	HMI_ParametriAsseJ_CicloFalda.Dec_Carico 		:= HMI_ParametriAsseJ_CicloFalda.Acc_Carico;
	HMI_ParametriAsseJ_CicloFalda.Dec_Vuoto  		:= HMI_ParametriAsseJ_CicloFalda.Acc_Vuoto;
	
	HMI_ParametriAsseK_CicloFalda.Dec_Carico 		:= HMI_ParametriAsseK_CicloFalda.Acc_Carico;
	HMI_ParametriAsseK_CicloFalda.Dec_Vuoto  		:= HMI_ParametriAsseK_CicloFalda.Acc_Vuoto;
	
	(* ASSE X *)
	ParametriProgramma_X_CicloFalda.Acc_Carico		:= AxisNominalPar_X.MaximumAcceleration * (HMI_ParametriAsseX_CicloFalda.Acc_Carico/100);
	ParametriProgramma_X_CicloFalda.Acc_Vuoto		:= AxisNominalPar_X.MaximumAcceleration * (HMI_ParametriAsseX_CicloFalda.Acc_Vuoto/100);
	ParametriProgramma_X_CicloFalda.Dec_Carico 		:= AxisNominalPar_X.MaximumDeceleration * (HMI_ParametriAsseX_CicloFalda.Dec_Carico/100);
	ParametriProgramma_X_CicloFalda.Dec_Vuoto  		:= AxisNominalPar_X.MaximumDeceleration * (HMI_ParametriAsseX_CicloFalda.Dec_Vuoto/100);
	ParametriProgramma_X_CicloFalda.Jerk_Carico  	:= AxisNominalPar_X.DefaultJerk * (HMI_ParametriAsseX_CicloFalda.Jerk_Carico/100);
	ParametriProgramma_X_CicloFalda.Jerk_Vuoto  	:= AxisNominalPar_X.DefaultJerk * (HMI_ParametriAsseX_CicloFalda.Jerk_Vuoto/100);
	ParametriProgramma_X_CicloFalda.Torque  		:= AxisNominalPar_X.DefaultTorque * (HMI_ParametriAsseX_CicloFalda.Torque/100);
	ParametriProgramma_X_CicloFalda.Vel_Carico  	:= AxisNominalPar_X.ReferenceVelocity * (HMI_ParametriAsseX_CicloFalda.Vel_Carico/100) * OverrideGlobaleCicloFalda;
	ParametriProgramma_X_CicloFalda.Vel_Ridotta  	:= AxisNominalPar_X.ReferenceVelocity * (HMI_ParametriAsseX_CicloFalda.Vel_Ridotta/100);// * OverrideGlobaleCicloFalda;
	ParametriProgramma_X_CicloFalda.Vel_Vuoto  		:= AxisNominalPar_X.ReferenceVelocity * (HMI_ParametriAsseX_CicloFalda.Vel_Vuoto/100) * OverrideGlobaleCicloAvuoto;
	(* ASSE Y *)
	ParametriProgramma_Y_CicloFalda.Acc_Carico		:= AxisNominalPar_Y.MaximumAcceleration * (HMI_ParametriAsseY_CicloFalda.Acc_Carico/100);
	ParametriProgramma_Y_CicloFalda.Acc_Vuoto		:= AxisNominalPar_Y.MaximumAcceleration * (HMI_ParametriAsseY_CicloFalda.Acc_Vuoto/100);
	ParametriProgramma_Y_CicloFalda.Dec_Carico 		:= AxisNominalPar_Y.MaximumDeceleration * (HMI_ParametriAsseY_CicloFalda.Dec_Carico/100);
	ParametriProgramma_Y_CicloFalda.Dec_Vuoto  		:= AxisNominalPar_Y.MaximumDeceleration * (HMI_ParametriAsseY_CicloFalda.Dec_Vuoto/100);
	ParametriProgramma_Y_CicloFalda.Jerk_Carico  	:= AxisNominalPar_Y.DefaultJerk * (HMI_ParametriAsseY_CicloFalda.Jerk_Carico/100);
	ParametriProgramma_Y_CicloFalda.Jerk_Vuoto  	:= AxisNominalPar_Y.DefaultJerk * (HMI_ParametriAsseY_CicloFalda.Jerk_Vuoto/100);
	ParametriProgramma_Y_CicloFalda.Torque  		:= AxisNominalPar_Y.DefaultTorque * (HMI_ParametriAsseY_CicloFalda.Torque/100);
	ParametriProgramma_Y_CicloFalda.Vel_Carico  	:= AxisNominalPar_Y.ReferenceVelocity * (HMI_ParametriAsseY_CicloFalda.Vel_Carico/100) * OverrideGlobaleCicloFalda;
	ParametriProgramma_Y_CicloFalda.Vel_Ridotta  	:= AxisNominalPar_Y.ReferenceVelocity * (HMI_ParametriAsseY_CicloFalda.Vel_Ridotta/100);// * OverrideGlobaleCicloFalda;
	ParametriProgramma_Y_CicloFalda.Vel_Vuoto  		:= AxisNominalPar_Y.ReferenceVelocity * (HMI_ParametriAsseY_CicloFalda.Vel_Vuoto/100) * OverrideGlobaleCicloAvuoto;
	(* ASSE Z *)
	ParametriProgramma_Z_CicloFalda.Acc_Carico		:= AxisNominalPar_Z.MaximumAcceleration * (HMI_ParametriAsseZ_CicloFalda.Acc_Carico/100);
	ParametriProgramma_Z_CicloFalda.Acc_Vuoto		:= AxisNominalPar_Z.MaximumAcceleration * (HMI_ParametriAsseZ_CicloFalda.Acc_Vuoto/100);
	ParametriProgramma_Z_CicloFalda.Dec_Carico 		:= AxisNominalPar_Z.MaximumDeceleration * (HMI_ParametriAsseZ_CicloFalda.Dec_Carico/100);
	ParametriProgramma_Z_CicloFalda.Dec_Vuoto  		:= AxisNominalPar_Z.MaximumDeceleration * (HMI_ParametriAsseZ_CicloFalda.Dec_Vuoto/100);
	ParametriProgramma_Z_CicloFalda.Jerk_Carico  	:= AxisNominalPar_Z.DefaultJerk * (HMI_ParametriAsseZ_CicloFalda.Jerk_Carico/100);
	ParametriProgramma_Z_CicloFalda.Jerk_Vuoto  	:= AxisNominalPar_Z.DefaultJerk * (HMI_ParametriAsseZ_CicloFalda.Jerk_Vuoto/100);
	ParametriProgramma_Z_CicloFalda.Torque  		:= AxisNominalPar_Z.DefaultTorque * (HMI_ParametriAsseZ_CicloFalda.Torque/100);
	ParametriProgramma_Z_CicloFalda.Vel_Carico  	:= AxisNominalPar_Z.ReferenceVelocity * (HMI_ParametriAsseZ_CicloFalda.Vel_Carico/100) * OverrideGlobaleCicloFalda;
	ParametriProgramma_Z_CicloFalda.Vel_Ridotta  	:= AxisNominalPar_Z.ReferenceVelocity * (HMI_ParametriAsseZ_CicloFalda.Vel_Ridotta/100); //* OverrideGlobaleCicloFalda;
	ParametriProgramma_Z_CicloFalda.Vel_Vuoto  		:= AxisNominalPar_Z.ReferenceVelocity * (HMI_ParametriAsseZ_CicloFalda.Vel_Vuoto/100) * OverrideGlobaleCicloAvuoto;
	(* ASSE J *)
	ParametriProgramma_J_CicloFalda.Acc_Carico		:= AxisNominalPar_J.MaximumAcceleration * (HMI_ParametriAsseJ_CicloFalda.Acc_Carico/100);
	ParametriProgramma_J_CicloFalda.Acc_Vuoto		:= AxisNominalPar_J.MaximumAcceleration * (HMI_ParametriAsseJ_CicloFalda.Acc_Vuoto/100);
	ParametriProgramma_J_CicloFalda.Dec_Carico 		:= AxisNominalPar_J.MaximumDeceleration * (HMI_ParametriAsseJ_CicloFalda.Dec_Carico/100);
	ParametriProgramma_J_CicloFalda.Dec_Vuoto  		:= AxisNominalPar_J.MaximumDeceleration * (HMI_ParametriAsseJ_CicloFalda.Dec_Vuoto/100);
	ParametriProgramma_J_CicloFalda.Jerk_Carico  	:= AxisNominalPar_J.DefaultJerk * (HMI_ParametriAsseJ_CicloFalda.Jerk_Carico/100);
	ParametriProgramma_J_CicloFalda.Jerk_Vuoto  	:= AxisNominalPar_J.DefaultJerk * (HMI_ParametriAsseJ_CicloFalda.Jerk_Vuoto/100);
	ParametriProgramma_J_CicloFalda.Torque  		:= AxisNominalPar_J.DefaultTorque * (HMI_ParametriAsseJ_CicloFalda.Torque/100);
	ParametriProgramma_J_CicloFalda.Vel_Carico  	:= AxisNominalPar_J.ReferenceVelocity * (HMI_ParametriAsseJ_CicloFalda.Vel_Carico/100);// * OverrideGlobaleCicloFalda;
	ParametriProgramma_J_CicloFalda.Vel_Ridotta  	:= AxisNominalPar_J.ReferenceVelocity * (HMI_ParametriAsseJ_CicloFalda.Vel_Ridotta/100);// * OverrideGlobaleCicloFalda;
	ParametriProgramma_J_CicloFalda.Vel_Vuoto  		:= AxisNominalPar_J.ReferenceVelocity * (HMI_ParametriAsseJ_CicloFalda.Vel_Vuoto/100);// * OverrideGlobaleCicloAvuoto;
	(* ASSE K *)
	(*
	ParametriProgramma_K_CicloFalda.Acc_Carico		:= AxisNominalPar_K.MaximumAcceleration * (HMI_ParametriAsseK_CicloFalda.Acc_Carico/100);
	ParametriProgramma_K_CicloFalda.Acc_Vuoto		:= AxisNominalPar_K.MaximumAcceleration * (HMI_ParametriAsseK_CicloFalda.Acc_Vuoto/100);
	ParametriProgramma_K_CicloFalda.Dec_Carico 		:= AxisNominalPar_K.MaximumDeceleration * (HMI_ParametriAsseK_CicloFalda.Dec_Carico/100);
	ParametriProgramma_K_CicloFalda.Dec_Vuoto  		:= AxisNominalPar_K.MaximumDeceleration * (HMI_ParametriAsseK_CicloFalda.Dec_Vuoto/100);
	ParametriProgramma_K_CicloFalda.Jerk_Carico  	:= AxisNominalPar_K.DefaultJerk * (HMI_ParametriAsseK_CicloFalda.Jerk_Carico/100);
	ParametriProgramma_K_CicloFalda.Jerk_Vuoto  	:= AxisNominalPar_K.DefaultJerk * (HMI_ParametriAsseK_CicloFalda.Jerk_Vuoto/100);
	//ParametriProgramma_K_CicloFalda.Torque  		:= Mission^.KPickTorque;//AxisNominalPar_K.DefaultTorque * (HMI_ParametriAsseK_CicloFalda.Torque/100);
	ParametriProgramma_K_CicloFalda.Vel_Carico  	:= AxisNominalPar_K.ReferenceVelocity * (HMI_ParametriAsseK_CicloFalda.Vel_Carico/100);// * OverrideGlobaleCicloFalda;
	ParametriProgramma_K_CicloFalda.Vel_Ridotta  	:= AxisNominalPar_K.ReferenceVelocity * (HMI_ParametriAsseK_CicloFalda.Vel_Ridotta/100);// * OverrideGlobaleCicloFalda;
	ParametriProgramma_K_CicloFalda.Vel_Vuoto  		:= AxisNominalPar_K.ReferenceVelocity * (HMI_ParametriAsseK_CicloFalda.Vel_Vuoto/100);// * OverrideGlobaleCicloAvuoto;
	*)
////////////////////////////////////////////////////////////////////////////////////////////////////////////////////////////////////////////////
//////////////////////////////////////////////////// CICLO PALLET //////////////////////////////////////////////////////////////////////////////
////////////////////////////////////////////////////////////////////////////////////////////////////////////////////////////////////////////////

	HMI_ParametriAsseX_CicloPallet.Dec_Carico 		:= HMI_ParametriAsseX_CicloPallet.Acc_Carico;
	HMI_ParametriAsseX_CicloPallet.Dec_Vuoto  		:= HMI_ParametriAsseX_CicloPallet.Acc_Vuoto;

	HMI_ParametriAsseY_CicloPallet.Dec_Carico 		:= HMI_ParametriAsseY_CicloPallet.Acc_Carico;
	HMI_ParametriAsseY_CicloPallet.Dec_Vuoto  		:= HMI_ParametriAsseY_CicloPallet.Acc_Vuoto;
		
	HMI_ParametriAsseZ_CicloPallet.Dec_Carico 		:= HMI_ParametriAsseZ_CicloPallet.Acc_Carico;
	HMI_ParametriAsseZ_CicloPallet.Dec_Vuoto  		:= HMI_ParametriAsseZ_CicloPallet.Acc_Vuoto;
	
	HMI_ParametriAsseJ_CicloPallet.Dec_Carico 		:= HMI_ParametriAsseJ_CicloPallet.Acc_Carico;
	HMI_ParametriAsseJ_CicloPallet.Dec_Vuoto  		:= HMI_ParametriAsseJ_CicloPallet.Acc_Vuoto;
	
	HMI_ParametriAsseK_CicloPallet.Dec_Carico 		:= HMI_ParametriAsseK_CicloPallet.Acc_Carico;
	HMI_ParametriAsseK_CicloPallet.Dec_Vuoto  		:= HMI_ParametriAsseK_CicloPallet.Acc_Vuoto;
	
	(* ASSE X *)
	ParametriProgramma_X_CicloPallet.Acc_Carico		:= AxisNominalPar_X.MaximumAcceleration * (HMI_ParametriAsseX_CicloPallet.Acc_Carico/100);
	ParametriProgramma_X_CicloPallet.Acc_Vuoto		:= AxisNominalPar_X.MaximumAcceleration * (HMI_ParametriAsseX_CicloPallet.Acc_Vuoto/100);
	ParametriProgramma_X_CicloPallet.Dec_Carico 	:= AxisNominalPar_X.MaximumDeceleration * (HMI_ParametriAsseX_CicloPallet.Dec_Carico/100);
	ParametriProgramma_X_CicloPallet.Dec_Vuoto  	:= AxisNominalPar_X.MaximumDeceleration * (HMI_ParametriAsseX_CicloPallet.Dec_Vuoto/100);
	ParametriProgramma_X_CicloPallet.Jerk_Carico  	:= AxisNominalPar_X.DefaultJerk * (HMI_ParametriAsseX_CicloPallet.Jerk_Carico/100);
	ParametriProgramma_X_CicloPallet.Jerk_Vuoto  	:= AxisNominalPar_X.DefaultJerk * (HMI_ParametriAsseX_CicloPallet.Jerk_Vuoto/100);
	ParametriProgramma_X_CicloPallet.Torque  		:= AxisNominalPar_X.DefaultTorque * (HMI_ParametriAsseX_CicloPallet.Torque/100);
	ParametriProgramma_X_CicloPallet.Vel_Carico  	:= AxisNominalPar_X.ReferenceVelocity * (HMI_ParametriAsseX_CicloPallet.Vel_Carico/100) * OverrideGlobaleCicloPallet;
	ParametriProgramma_X_CicloPallet.Vel_Ridotta  	:= AxisNominalPar_X.ReferenceVelocity * (HMI_ParametriAsseX_CicloPallet.Vel_Ridotta/100);
	ParametriProgramma_X_CicloPallet.Vel_Vuoto  	:= AxisNominalPar_X.ReferenceVelocity * (HMI_ParametriAsseX_CicloPallet.Vel_Vuoto/100) * OverrideGlobaleCicloPallet;
	(* ASSE Y *)
	ParametriProgramma_Y_CicloPallet.Acc_Carico		:= AxisNominalPar_Y.MaximumAcceleration * (HMI_ParametriAsseY_CicloPallet.Acc_Carico/100);
	ParametriProgramma_Y_CicloPallet.Acc_Vuoto		:= AxisNominalPar_Y.MaximumAcceleration * (HMI_ParametriAsseY_CicloPallet.Acc_Vuoto/100);
	ParametriProgramma_Y_CicloPallet.Dec_Carico 	:= AxisNominalPar_Y.MaximumDeceleration * (HMI_ParametriAsseY_CicloPallet.Dec_Carico/100);
	ParametriProgramma_Y_CicloPallet.Dec_Vuoto  	:= AxisNominalPar_Y.MaximumDeceleration * (HMI_ParametriAsseY_CicloPallet.Dec_Vuoto/100);
	ParametriProgramma_Y_CicloPallet.Jerk_Carico  	:= AxisNominalPar_Y.DefaultJerk * (HMI_ParametriAsseY_CicloPallet.Jerk_Carico/100);
	ParametriProgramma_Y_CicloPallet.Jerk_Vuoto  	:= AxisNominalPar_Y.DefaultJerk * (HMI_ParametriAsseY_CicloPallet.Jerk_Vuoto/100);
	ParametriProgramma_Y_CicloPallet.Torque  		:= AxisNominalPar_Y.DefaultTorque * (HMI_ParametriAsseY_CicloPallet.Torque/100);
	ParametriProgramma_Y_CicloPallet.Vel_Carico  	:= AxisNominalPar_Y.ReferenceVelocity * (HMI_ParametriAsseY_CicloPallet.Vel_Carico/100) * OverrideGlobaleCicloPallet;
	ParametriProgramma_Y_CicloPallet.Vel_Ridotta  	:= AxisNominalPar_Y.ReferenceVelocity * (HMI_ParametriAsseY_CicloPallet.Vel_Ridotta/100);// * OverrideGlobaleCicloPallet;
	ParametriProgramma_Y_CicloPallet.Vel_Vuoto  	:= AxisNominalPar_Y.ReferenceVelocity * (HMI_ParametriAsseY_CicloPallet.Vel_Vuoto/100) * OverrideGlobaleCicloAvuoto;
	(* ASSE Z *)
	ParametriProgramma_Z_CicloPallet.Acc_Carico		:= AxisNominalPar_Z.MaximumAcceleration * (HMI_ParametriAsseZ_CicloPallet.Acc_Carico/100);
	ParametriProgramma_Z_CicloPallet.Acc_Vuoto		:= AxisNominalPar_Z.MaximumAcceleration * (HMI_ParametriAsseZ_CicloPallet.Acc_Vuoto/100);
	ParametriProgramma_Z_CicloPallet.Dec_Carico 	:= AxisNominalPar_Z.MaximumDeceleration * (HMI_ParametriAsseZ_CicloPallet.Dec_Carico/100);
	ParametriProgramma_Z_CicloPallet.Dec_Vuoto  	:= AxisNominalPar_Z.MaximumDeceleration * (HMI_ParametriAsseZ_CicloPallet.Dec_Vuoto/100);
	ParametriProgramma_Z_CicloPallet.Jerk_Carico  	:= AxisNominalPar_Z.DefaultJerk * (HMI_ParametriAsseZ_CicloPallet.Jerk_Carico/100);
	ParametriProgramma_Z_CicloPallet.Jerk_Vuoto  	:= AxisNominalPar_Z.DefaultJerk * (HMI_ParametriAsseZ_CicloPallet.Jerk_Vuoto/100);
	ParametriProgramma_Z_CicloPallet.Torque  		:= AxisNominalPar_Z.DefaultTorque * (HMI_ParametriAsseZ_CicloPallet.Torque/100);
	ParametriProgramma_Z_CicloPallet.Vel_Carico  	:= AxisNominalPar_Z.ReferenceVelocity * (HMI_ParametriAsseZ_CicloPallet.Vel_Carico/100) * OverrideGlobaleCicloPallet;
	ParametriProgramma_Z_CicloPallet.Vel_Ridotta  	:= AxisNominalPar_Z.ReferenceVelocity * (HMI_ParametriAsseZ_CicloPallet.Vel_Ridotta/100);// * OverrideGlobaleCicloPallet;
	ParametriProgramma_Z_CicloPallet.Vel_Vuoto  	:= AxisNominalPar_Z.ReferenceVelocity * (HMI_ParametriAsseZ_CicloPallet.Vel_Vuoto/100) * OverrideGlobaleCicloAvuoto;
	(* ASSE J *)
	ParametriProgramma_J_CicloPallet.Acc_Carico		:= AxisNominalPar_J.MaximumAcceleration * (HMI_ParametriAsseJ_CicloPallet.Acc_Carico/100);
	ParametriProgramma_J_CicloPallet.Acc_Vuoto		:= AxisNominalPar_J.MaximumAcceleration * (HMI_ParametriAsseJ_CicloPallet.Acc_Vuoto/100);
	ParametriProgramma_J_CicloPallet.Dec_Carico 	:= AxisNominalPar_J.MaximumDeceleration * (HMI_ParametriAsseJ_CicloPallet.Dec_Carico/100);
	ParametriProgramma_J_CicloPallet.Dec_Vuoto  	:= AxisNominalPar_J.MaximumDeceleration * (HMI_ParametriAsseJ_CicloPallet.Dec_Vuoto/100);
	ParametriProgramma_J_CicloPallet.Jerk_Carico  	:= AxisNominalPar_J.DefaultJerk * (HMI_ParametriAsseJ_CicloPallet.Jerk_Carico/100);
	ParametriProgramma_J_CicloPallet.Jerk_Vuoto  	:= AxisNominalPar_J.DefaultJerk * (HMI_ParametriAsseJ_CicloPallet.Jerk_Vuoto/100);
	ParametriProgramma_J_CicloPallet.Torque  		:= AxisNominalPar_J.DefaultTorque * (HMI_ParametriAsseJ_CicloPallet.Torque/100);
	ParametriProgramma_J_CicloPallet.Vel_Carico  	:= AxisNominalPar_J.ReferenceVelocity * (HMI_ParametriAsseJ_CicloPallet.Vel_Carico/100);// * OverrideGlobaleCicloPallet;
	ParametriProgramma_J_CicloPallet.Vel_Ridotta  	:= AxisNominalPar_J.ReferenceVelocity * (HMI_ParametriAsseJ_CicloPallet.Vel_Ridotta/100);// * OverrideGlobaleCicloPallet;
	ParametriProgramma_J_CicloPallet.Vel_Vuoto  	:= AxisNominalPar_J.ReferenceVelocity * (HMI_ParametriAsseJ_CicloPallet.Vel_Vuoto/100);// * OverrideGlobaleCicloAvuoto;
	(* ASSE K *)
	(*
	ParametriProgramma_K_CicloPallet.Acc_Carico		:= AxisNominalPar_K.MaximumAcceleration * (HMI_ParametriAsseK_CicloPallet.Acc_Carico/100);
	ParametriProgramma_K_CicloPallet.Acc_Vuoto		:= AxisNominalPar_K.MaximumAcceleration * (HMI_ParametriAsseK_CicloPallet.Acc_Vuoto/100);
	ParametriProgramma_K_CicloPallet.Dec_Carico 	:= AxisNominalPar_K.MaximumDeceleration * (HMI_ParametriAsseK_CicloPallet.Dec_Carico/100);
	ParametriProgramma_K_CicloPallet.Dec_Vuoto  	:= AxisNominalPar_K.MaximumDeceleration * (HMI_ParametriAsseK_CicloPallet.Dec_Vuoto/100);
	ParametriProgramma_K_CicloPallet.Jerk_Carico  	:= AxisNominalPar_K.DefaultJerk * (HMI_ParametriAsseK_CicloPallet.Jerk_Carico/100);
	ParametriProgramma_K_CicloPallet.Jerk_Vuoto  	:= AxisNominalPar_K.DefaultJerk * (HMI_ParametriAsseK_CicloPallet.Jerk_Vuoto/100);
	//ParametriProgramma_K_CicloPallet.Torque  		:= Mission^.KPickTorque;//AxisNominalPar_K.DefaultTorque * (HMI_ParametriAsseK_CicloPallet.Torque/100);
	ParametriProgramma_K_CicloPallet.Vel_Carico  	:= AxisNominalPar_K.ReferenceVelocity * (HMI_ParametriAsseK_CicloPallet.Vel_Carico/100);// * OverrideGlobaleCicloPallet;
	ParametriProgramma_K_CicloPallet.Vel_Ridotta  	:= AxisNominalPar_K.ReferenceVelocity * (HMI_ParametriAsseK_CicloPallet.Vel_Ridotta/100);// * OverrideGlobaleCicloPallet;
	ParametriProgramma_K_CicloPallet.Vel_Vuoto  	:= AxisNominalPar_K.ReferenceVelocity * (HMI_ParametriAsseK_CicloPallet.Vel_Vuoto/100);// * OverrideGlobaleCicloAvuoto;
	*)
////////////////////////////////////////////////////////////////////////////////////////////////////////////////////////////////////////////////
//////////////////////////////////////////////////// CICLO PACCO //////////////////////////////////////////////////////////////////////////////
////////////////////////////////////////////////////////////////////////////////////////////////////////////////////////////////////////////////


	HMI_ParametriAsseX_CicloPacco.Acc_Carico	:= MAX(1,HMI_ParametriAsseX_CicloPacco.Acc_Carico);
	HMI_ParametriAsseX_CicloPacco.Acc_Vuoto		:= MAX(1,HMI_ParametriAsseX_CicloPacco.Acc_Vuoto); 
																				 
	HMI_ParametriAsseY_CicloPacco.Acc_Carico	:= MAX(1,HMI_ParametriAsseY_CicloPacco.Acc_Carico);
	HMI_ParametriAsseY_CicloPacco.Acc_Vuoto		:= MAX(1,HMI_ParametriAsseY_CicloPacco.Acc_Vuoto); 
																				 
	HMI_ParametriAsseZ_CicloPacco.Acc_Carico	:= MAX(1,HMI_ParametriAsseZ_CicloPacco.Acc_Carico);
	HMI_ParametriAsseZ_CicloPacco.Acc_Vuoto		:= MAX(1,HMI_ParametriAsseZ_CicloPacco.Acc_Vuoto); 
																				 
	HMI_ParametriAsseJ_CicloPacco.Acc_Carico	:= MAX(1,HMI_ParametriAsseJ_CicloPacco.Acc_Carico);
	HMI_ParametriAsseJ_CicloPacco.Acc_Vuoto		:= MAX(1,HMI_ParametriAsseJ_CicloPacco.Acc_Vuoto); 
																			     
	HMI_ParametriAsseK_CicloPacco.Acc_Carico	:= MAX(1,HMI_ParametriAsseK_CicloPacco.Acc_Carico);
	HMI_ParametriAsseK_CicloPacco.Acc_Vuoto		:= MAX(1,HMI_ParametriAsseK_CicloPacco.Acc_Vuoto); 
                                                                                 
	HMI_ParametriAsseX_CicloPacco.Vel_Carico	:= MAX(1,HMI_ParametriAsseX_CicloPacco.Vel_Carico);	
	HMI_ParametriAsseX_CicloPacco.Vel_Ridotta  	:= MAX(1,HMI_ParametriAsseX_CicloPacco.Vel_Ridotta);
	

	HMI_ParametriAsseX_CicloPacco.Dec_Carico 		:= HMI_ParametriAsseX_CicloPacco.Acc_Carico;
	HMI_ParametriAsseX_CicloPacco.Dec_Vuoto  		:= HMI_ParametriAsseX_CicloPacco.Acc_Vuoto;

	HMI_ParametriAsseY_CicloPacco.Dec_Carico 		:= HMI_ParametriAsseY_CicloPacco.Acc_Carico;
	HMI_ParametriAsseY_CicloPacco.Dec_Vuoto  		:= HMI_ParametriAsseY_CicloPacco.Acc_Vuoto;
		
	HMI_ParametriAsseZ_CicloPacco.Dec_Carico 		:= HMI_ParametriAsseZ_CicloPacco.Acc_Carico;
	HMI_ParametriAsseZ_CicloPacco.Dec_Vuoto  		:= HMI_ParametriAsseZ_CicloPacco.Acc_Vuoto;
	
	HMI_ParametriAsseJ_CicloPacco.Dec_Carico 		:= HMI_ParametriAsseJ_CicloPacco.Acc_Carico;
	HMI_ParametriAsseJ_CicloPacco.Dec_Vuoto  		:= HMI_ParametriAsseJ_CicloPacco.Acc_Vuoto;
	
	HMI_ParametriAsseK_CicloPacco.Dec_Carico 		:= HMI_ParametriAsseK_CicloPacco.Acc_Carico;
	HMI_ParametriAsseK_CicloPacco.Dec_Vuoto  		:= HMI_ParametriAsseK_CicloPacco.Acc_Vuoto;

	(* ASSE X *)
	ParametriProgramma_X_CicloLastra.Acc_Carico		:= AxisNominalPar_X.MaximumAcceleration * (HMI_ParametriAsseX_CicloPacco.Acc_Carico/100);
	ParametriProgramma_X_CicloLastra.Acc_Vuoto		:= AxisNominalPar_X.MaximumAcceleration * (HMI_ParametriAsseX_CicloPacco.Acc_Vuoto/100);
	ParametriProgramma_X_CicloLastra.Dec_Carico 	:= AxisNominalPar_X.MaximumDeceleration * (HMI_ParametriAsseX_CicloPacco.Dec_Carico/100);
	ParametriProgramma_X_CicloLastra.Dec_Vuoto  	:= AxisNominalPar_X.MaximumDeceleration * (HMI_ParametriAsseX_CicloPacco.Dec_Vuoto/100);
	ParametriProgramma_X_CicloLastra.Jerk_Carico  	:= AxisNominalPar_X.DefaultJerk * (HMI_ParametriAsseX_CicloPacco.Jerk_Carico/100);
	ParametriProgramma_X_CicloLastra.Jerk_Vuoto  	:= AxisNominalPar_X.DefaultJerk * (HMI_ParametriAsseX_CicloPacco.Jerk_Vuoto/100);
	ParametriProgramma_X_CicloLastra.Torque  		:= AxisNominalPar_X.DefaultTorque * (HMI_ParametriAsseX_CicloPacco.Torque/100);
	//IF DepositoPaccoInLenta THEN
	//	ParametriProgramma_X_CicloLastra.Vel_Carico  := AxisNominalPar_X.ReferenceVelocity * (HMI_ParametriAsseX_CicloPacco.Vel_Carico/100) * OverrideGlobaleCicloPacco * (HMI_VelocitaDepositoPrimoPaccoInLenta/100);
	//ELSE
		ParametriProgramma_X_CicloLastra.Vel_Carico  := AxisNominalPar_X.ReferenceVelocity * (HMI_ParametriAsseX_CicloPacco.Vel_Carico/100) * OverrideGlobaleCicloPacco;
	//END_IF
	ParametriProgramma_X_CicloLastra.Vel_Ridotta  	:= AxisNominalPar_X.ReferenceVelocity * (HMI_ParametriAsseX_CicloPacco.Vel_Ridotta/100);// * OverrideGlobaleCicloPacco;
	ParametriProgramma_X_CicloLastra.Vel_Vuoto  		:= AxisNominalPar_X.ReferenceVelocity * (HMI_ParametriAsseX_CicloPacco.Vel_Vuoto/100) * OverrideGlobaleCicloAvuoto;
	(* ASSE Y *)
	ParametriProgramma_Y_CicloLastra.Acc_Carico		:= AxisNominalPar_Y.MaximumAcceleration * (HMI_ParametriAsseY_CicloPacco.Acc_Carico/100);
	ParametriProgramma_Y_CicloLastra.Acc_Vuoto		:= AxisNominalPar_Y.MaximumAcceleration * (HMI_ParametriAsseY_CicloPacco.Acc_Vuoto/100);
	ParametriProgramma_Y_CicloLastra.Dec_Carico 		:= AxisNominalPar_Y.MaximumDeceleration * (HMI_ParametriAsseY_CicloPacco.Dec_Carico/100);
	ParametriProgramma_Y_CicloLastra.Dec_Vuoto  		:= AxisNominalPar_Y.MaximumDeceleration * (HMI_ParametriAsseY_CicloPacco.Dec_Vuoto/100);
	ParametriProgramma_Y_CicloLastra.Jerk_Carico  	:= AxisNominalPar_Y.DefaultJerk * (HMI_ParametriAsseY_CicloPacco.Jerk_Carico/100);
	ParametriProgramma_Y_CicloLastra.Jerk_Vuoto  	:= AxisNominalPar_Y.DefaultJerk * (HMI_ParametriAsseY_CicloPacco.Jerk_Vuoto/100);
	ParametriProgramma_Y_CicloLastra.Torque  		:= AxisNominalPar_Y.DefaultTorque * (HMI_ParametriAsseY_CicloPacco.Torque/100);
	//IF DepositoPaccoInLenta THEN
	//	ParametriProgramma_Y_CicloLastra.Vel_Carico  	:= AxisNominalPar_Y.ReferenceVelocity * (HMI_ParametriAsseY_CicloPacco.Vel_Carico/100) * OverrideGlobaleCicloPacco * (HMI_VelocitaDepositoPrimoPaccoInLenta/100);
	//ELSE
		ParametriProgramma_Y_CicloLastra.Vel_Carico  	:= AxisNominalPar_Y.ReferenceVelocity * (HMI_ParametriAsseY_CicloPacco.Vel_Carico/100) * OverrideGlobaleCicloPacco;
	//END_IF
	ParametriProgramma_Y_CicloLastra.Vel_Ridotta  	:= AxisNominalPar_Y.ReferenceVelocity * (HMI_ParametriAsseY_CicloPacco.Vel_Ridotta/100);// * OverrideGlobaleCicloPacco;
	ParametriProgramma_Y_CicloLastra.Vel_Vuoto  		:= AxisNominalPar_Y.ReferenceVelocity * (HMI_ParametriAsseY_CicloPacco.Vel_Vuoto/100) * OverrideGlobaleCicloAvuoto;
	(* ASSE Z *)
	ParametriProgramma_Z_CicloLastra.Acc_Carico		:= AxisNominalPar_Z.MaximumAcceleration * (HMI_ParametriAsseZ_CicloPacco.Acc_Carico/100);
	ParametriProgramma_Z_CicloLastra.Acc_Vuoto		:= AxisNominalPar_Z.MaximumAcceleration * (HMI_ParametriAsseZ_CicloPacco.Acc_Vuoto/100);
	ParametriProgramma_Z_CicloLastra.Dec_Carico 		:= AxisNominalPar_Z.MaximumDeceleration * (HMI_ParametriAsseZ_CicloPacco.Dec_Carico/100);
	ParametriProgramma_Z_CicloLastra.Dec_Vuoto  		:= AxisNominalPar_Z.MaximumDeceleration * (HMI_ParametriAsseZ_CicloPacco.Dec_Vuoto/100);
	ParametriProgramma_Z_CicloLastra.Jerk_Carico  	:= AxisNominalPar_Z.DefaultJerk * (HMI_ParametriAsseZ_CicloPacco.Jerk_Carico/100);
	ParametriProgramma_Z_CicloLastra.Jerk_Vuoto  	:= AxisNominalPar_Z.DefaultJerk * (HMI_ParametriAsseZ_CicloPacco.Jerk_Vuoto/100);
	ParametriProgramma_Z_CicloLastra.Torque  		:= AxisNominalPar_Z.DefaultTorque * (HMI_ParametriAsseZ_CicloPacco.Torque/100);
	IF DepositoPaccoInLenta THEN
		ParametriProgramma_Z_CicloLastra.Vel_Carico  	:= AxisNominalPar_Z.ReferenceVelocity * (HMI_ParametriAsseZ_CicloPacco.Vel_Carico/100) * OverrideGlobaleCicloPacco * (HMI_VelocitaDepositoPrimoPaccoInLenta/100);
	ELSE
		ParametriProgramma_Z_CicloLastra.Vel_Carico  	:= AxisNominalPar_Z.ReferenceVelocity * (HMI_ParametriAsseZ_CicloPacco.Vel_Carico/100) * OverrideGlobaleCicloPacco;		
	END_IF
	ParametriProgramma_Z_CicloLastra.Vel_Ridotta  	:= AxisNominalPar_Z.ReferenceVelocity * (HMI_ParametriAsseZ_CicloPacco.Vel_Ridotta/100);// * OverrideGlobaleCicloPacco;
	ParametriProgramma_Z_CicloLastra.Vel_Vuoto  		:= AxisNominalPar_Z.ReferenceVelocity * (HMI_ParametriAsseZ_CicloPacco.Vel_Vuoto/100) * OverrideGlobaleCicloAvuoto;
	(* ASSE J *)
	ParametriProgramma_J_CicloLastra.Acc_Carico		:= AxisNominalPar_J.MaximumAcceleration * (HMI_ParametriAsseJ_CicloPacco.Acc_Carico/100);
	ParametriProgramma_J_CicloLastra.Acc_Vuoto		:= AxisNominalPar_J.MaximumAcceleration * (HMI_ParametriAsseJ_CicloPacco.Acc_Vuoto/100);
	ParametriProgramma_J_CicloLastra.Dec_Carico 		:= AxisNominalPar_J.MaximumDeceleration * (HMI_ParametriAsseJ_CicloPacco.Dec_Carico/100);
	ParametriProgramma_J_CicloLastra.Dec_Vuoto  		:= AxisNominalPar_J.MaximumDeceleration * (HMI_ParametriAsseJ_CicloPacco.Dec_Vuoto/100);
	ParametriProgramma_J_CicloLastra.Jerk_Carico  	:= AxisNominalPar_J.DefaultJerk * (HMI_ParametriAsseJ_CicloPacco.Jerk_Carico/100);
	ParametriProgramma_J_CicloLastra.Jerk_Vuoto  	:= AxisNominalPar_J.DefaultJerk * (HMI_ParametriAsseJ_CicloPacco.Jerk_Vuoto/100);
	ParametriProgramma_J_CicloLastra.Torque  		:= AxisNominalPar_J.DefaultTorque * (HMI_ParametriAsseJ_CicloPacco.Torque/100);
	//IF DepositoPaccoInLenta THEN
	//	ParametriProgramma_J_CicloLastra.Vel_Carico  	:= AxisNominalPar_J.ReferenceVelocity * (HMI_ParametriAsseJ_CicloPacco.Vel_Carico/100) * OverrideGlobaleCicloPacco * (HMI_VelocitaDepositoPrimoPaccoInLenta/100);
	//ELSE
		ParametriProgramma_J_CicloLastra.Vel_Carico  	:= AxisNominalPar_J.ReferenceVelocity * (HMI_ParametriAsseJ_CicloPacco.Vel_Carico/100);// * OverrideGlobaleCicloPacco;		
	//END_IF
	ParametriProgramma_J_CicloLastra.Vel_Ridotta  	:= AxisNominalPar_J.ReferenceVelocity * (HMI_ParametriAsseJ_CicloPacco.Vel_Ridotta/100);// * OverrideGlobaleCicloPacco;
	ParametriProgramma_J_CicloLastra.Vel_Vuoto  		:= AxisNominalPar_J.ReferenceVelocity * (HMI_ParametriAsseJ_CicloPacco.Vel_Vuoto/100);// * OverrideGlobaleCicloAvuoto;
	(* ASSE K *)
	(*ParametriProgramma_K_CicloLastra.Acc_Carico		:= AxisNominalPar_K.MaximumAcceleration * (HMI_ParametriAsseK_CicloPacco.Acc_Carico/100);
	ParametriProgramma_K_CicloLastra.Acc_Vuoto		:= AxisNominalPar_K.MaximumAcceleration * (HMI_ParametriAsseK_CicloPacco.Acc_Vuoto/100);
	ParametriProgramma_K_CicloLastra.Dec_Carico 		:= AxisNominalPar_K.MaximumDeceleration * (HMI_ParametriAsseK_CicloPacco.Dec_Carico/100);
	ParametriProgramma_K_CicloLastra.Dec_Vuoto  		:= AxisNominalPar_K.MaximumDeceleration * (HMI_ParametriAsseK_CicloPacco.Dec_Vuoto/100);
	ParametriProgramma_K_CicloLastra.Jerk_Carico  	:= AxisNominalPar_K.DefaultJerk * (HMI_ParametriAsseK_CicloPacco.Jerk_Carico/100);
	ParametriProgramma_K_CicloLastra.Jerk_Vuoto  	:= AxisNominalPar_K.DefaultJerk * (HMI_ParametriAsseK_CicloPacco.Jerk_Vuoto/100);
	//ParametriProgramma_K_CicloLastra.Torque  		:= Mission^.KPickTorque;//AxisNominalPar_K.DefaultTorque * (HMI_ParametriAsseK_CicloPacco.Torque/100);
	ParametriProgramma_K_CicloLastra.Vel_Carico  	:= AxisNominalPar_K.ReferenceVelocity * (HMI_ParametriAsseK_CicloPacco.Vel_Carico/100);//* OverrideGlobaleCicloPacco;
	ParametriProgramma_K_CicloLastra.Vel_Ridotta  	:= AxisNominalPar_K.ReferenceVelocity * (HMI_ParametriAsseK_CicloPacco.Vel_Ridotta/100);// * OverrideGlobaleCicloPacco;
	ParametriProgramma_K_CicloLastra.Vel_Vuoto  		:= AxisNominalPar_K.ReferenceVelocity * (HMI_ParametriAsseK_CicloPacco.Vel_Vuoto/100);//* OverrideGlobaleCicloAvuoto;
	*)

TFCalcoloVelocita := TRUE;

END_FUNCTION

// ---- POUs/TFPalletizerDataTF/TFCalcoloOverrideDinamico.TcPOU
FUNCTION TFCalcoloOverrideDinamico : REAL
VAR_INPUT
	NUltimiTrasportiOccupati : UINT;
	Overide_Dinamico : Overide_Dinamico;
END_VAR
VAR
	i : uint;
END_VAR


FOR i:= 1 TO MAXSOGLIEOVERRIDE DO
	IF NUltimiTrasportiOccupati >= Overide_Dinamico.NTrasportiOccupati[i] THEN
		TFCalcoloOverrideDinamico := Overide_Dinamico.Override[i];
		RETURN;
	END_IF
END_FOR

END_FUNCTION

// ---- POUs/TFPalletizerDataTF/TFFuoriIngombroVerticaleOK.TcPOU
FUNCTION TFFuoriIngombroVerticaleOK : BOOL
VAR_INPUT
	QuotaAsseZ : LREAL;
	Mission : POINTER TO TFMachinePalletizer_Mission;
END_VAR
VAR
END_VAR

(* Controllo Asse Z Fuori Ingombro *)
CASE Mission^.TPick OF
	TPICK_LAYER:
					IF QuotaAsseZ >= QuotaFuoriIngombro_Z_AVUOTO OR 
					QuotaAsseZ >= QuotaFuoriIngombro_Z_ConFALDA THEN
						TFFuoriIngombroVerticaleOK := TRUE;
					ELSE
						TFFuoriIngombroVerticaleOK := FALSE;
					END_IF
	TPICK_PACK :
					IF QuotaAsseZ >= QuotaFuoriIngombro_Z_AVUOTO OR 
					QuotaAsseZ >= QuotaFuoriIngombro_Z_ConPEZZO THEN
						TFFuoriIngombroVerticaleOK := TRUE;
					ELSE
						TFFuoriIngombroVerticaleOK := FALSE;
					END_IF
	TPICK_PALLET:
					IF QuotaAsseZ >= QuotaFuoriIngombro_Z_AVUOTO OR 
					QuotaAsseZ >= QuotaFuoriIngombro_Z_ConPALLET THEN
						TFFuoriIngombroVerticaleOK := TRUE;
					ELSE
						TFFuoriIngombroVerticaleOK := FALSE;
					END_IF
					
	TPICK_NOT_DEFINED:
					IF QuotaAsseZ >= QuotaFuoriIngombro_Z_AVUOTO OR 
					QuotaAsseZ >= QuotaFuoriIngombro_Z_ConPEZZO OR 
					QuotaAsseZ >= QuotaFuoriIngombro_Z_ConPALLET OR
					QuotaAsseZ >= QuotaFuoriIngombro_Z_ConFALDA THEN
						TFFuoriIngombroVerticaleOK := TRUE;
					ELSE
						TFFuoriIngombroVerticaleOK := FALSE;
					END_IF
					
	TPICK_LASTRA:
					IF QuotaAsseZ >= QuotaFuoriIngombro_Z_AVUOTO OR 
					QuotaAsseZ >= QuotaFuoriIngombro_Z_ConPEZZO THEN
						TFFuoriIngombroVerticaleOK := TRUE;
					ELSE
						TFFuoriIngombroVerticaleOK := FALSE;
					END_IF
					
	TPICK_QUADROTTA:
					IF QuotaAsseZ >= QuotaFuoriIngombro_Z_AVUOTO OR 
					QuotaAsseZ >= QuotaFuoriIngombro_Z_ConPEZZO THEN
						TFFuoriIngombroVerticaleOK := TRUE;
					ELSE
						TFFuoriIngombroVerticaleOK := FALSE;
					END_IF
					
					
					
					
					
END_CASE

END_FUNCTION

// ---- POUs/TFModules/Moduli TF/TFModulePalletizer_Aspirazione.TcPOU

FUNCTION_BLOCK TFModulePalletizer_Aspirazione
VAR_INPUT
	Cmd : CommandBuffer;
	Cfg : Config;
	IN : Module_Palletizer_Aspirazione_IN;
	
	ManCmd : Module_Palletizer_Aspirazione_ManCmd;
	
END_VAR
VAR_OUTPUT
	CmdExe : CommandExe;
	CmdExd : CommandExe;
	CmdNext : Command;
	CmdLog : CommandLog;
	ProgramLog : ProgrammaLog; 
	State : State;
	StateLog : StateLog;
	Error : Error;
	ErrorLog : ErrorLog;
	Warning : Warning;
	WarningLog : WarningLog;
	OUT : Module_Palletizer_Aspirazione_OUT;
END_VAR
VAR
	Power : UINT;
	Init : BOOL;
	Timer : REAL;
	Timeout : REAL;
	TimerAspirazione : REAL;
	ParametersArray : ParametersArray;
	MAN_Actuator : UINT;
	MAN_Cmd : UINT;
END_VAR

IF NOT Init THEN
	TFCommandBufferClear(ADR(Cmd));
	TFCommandClear(ADR(CmdNext));
	TFCommandExeClear(ADR(CmdExe));
	TFStateUpdate(ADR(State),StateNOP);
	TFErrorClear(ADR(Error));
	TFWarningClear(ADR(Warning));
	Init := TRUE;
	CmdExe.Code := 1;
END_IF

(* Generic Timer - Add here all your Timers *)
TFTimerCall(ADR(Timer),Cfg.TimeBase);
TFTimerCall(ADR(Timeout),Cfg.TimeBase);
TFTimerCall(ADR(TimerAspirazione),Cfg.TimeBase);
(* External To Buffered Command *)
TFCommandToNext(ADR(Cmd),ADR(CmdNext),ADR(CmdExe),ADR(Cfg),ADR(Error),ADR(ErrorLog),ADR(State));

(* Buffered To Exe Command *)
TFCommandToExecution(ADR(CmdNext),ADR(CmdExe),ADR(Error),ADR(ErrorLog),ADR(State),ADR(CmdLog));

(* Exe Command *)
CASE CmdExe.Code OF

	(* ******************************************************************************************************** *)
	(* Nop  *)
	(* ******************************************************************************************************** *)
	CmdNOP:	;
	
	1: TFStateUpdate(ADR(State),CmdNOP);

	(* ******************************************************************************************************** *)
	(* Stop *)
	(* ******************************************************************************************************** *)
	CmdSTOP:
		CASE CmdExe.CmdCase OF
			
			(* Case 0 *)
			0: 	TFStateUpdate(ADR(State),StateSTOP_RUN);
				TFTimerSet(ADR(Timeout),500,TRUE);
				TFCommandCase(ADR(CmdExe),1,CommandCase_INC);

			(* Case 1 - Clear All Commands*)
			1:	
				TFCommandCase(ADR(CmdExe),100,CommandCase_JMP);
			(* Case 100 *)
			100:TFStateUpdate(ADR(State),StateSTOP_END);
				TFCommandExeClear(ADR(CmdExe));

			ELSE
				TFError(ErrNOCMDCASE,ErrNULL,ADR(CmdExe),ADR(State),ADR(Error),ADR(ErrorLog));
		END_CASE;
	
	(* ******************************************************************************************************** *)
	(* Error Reset *)
	(* ******************************************************************************************************** *)
	CmdRESET:
		CASE CmdExe.CmdCase OF

			(* Case 0 *)
			0: 	TFStateUpdate(ADR(State),StateRESET_RUN);
				TFTimerSet(ADR(Timeout),2000,TRUE);
				TFCommandCase(ADR(CmdExe),1,CommandCase_INC);
			
			(* Case 1 *)
			1: TFCommandCase(ADR(CmdExe),99,CommandCase_JMP);

			
			(* Case 99 *)
			99:	TFErrorClear(ADR(Error));
				TFWarningClear(ADR(Warning));
				TFCommandCase(ADR(CmdExe),100,CommandCase_JMP);

			(* Case 100 *)
			100:TFStateUpdate(ADR(State),StateRESET_END);
				TFCommandExeClear(ADR(CmdExe));

			ELSE
				TFError(ErrNOCMDCASE,ErrNULL,ADR(CmdExe),ADR(State),ADR(Error),ADR(ErrorLog));
		END_CASE;
	
	(* ******************************************************************************************************** *)
	(* Power *)
	(* ******************************************************************************************************** *)
	CmdPOWER:
		CASE CmdExe.CmdCase OF
			
			(* Case 0 *)
			0: 	TFStateUpdate(ADR(State),StatePOWER_RUN);
				TFTimerSet(ADR(Timeout),500,TRUE);

			1: TFCommandCase(ADR(CmdExe),100,CommandCase_JMP);
			(* Case 100 *)
			100:TFStateUpdate(ADR(State),StatePOWER_END);
				TFCommandExeClear(ADR(CmdExe));

			ELSE
				TFError(ErrNOCMDCASE,ErrNULL,ADR(CmdExe),ADR(State),ADR(Error),ADR(ErrorLog));
		END_CASE
	
	(* ******************************************************************************************************** *)
	(* Home *)
	(* ******************************************************************************************************** *)
	CmdHOME:
		CASE CmdExe.CmdCase OF

			(* Case 0 *)
			0: 	TFStateUpdate(ADR(State),StateHOME_RUN);
				TFTimerSet(ADR(Timeout),30000,TRUE);
				TFCommandCase(ADR(CmdExe),1,CommandCase_INC);

			(* Case 1 - Disattivazione + Salita Ventose*)
			1: OUT.EV_Suction := FALSE;
				OUT.EV_SuctionCupsDown := FALSE;
				OUT.EV_SuctionCupsUP := TRUE;
				TFCommandCase(ADR(CmdExe),100,CommandCase_JMP);
	
			(* Case 100 *)
			100:TFStateUpdate(ADR(State),StateHOME_END);
				TFCommandExeClear(ADR(CmdExe));

			ELSE
				TFError(ErrNOCMDCASE,ErrNULL,ADR(CmdExe),ADR(State),ADR(Error),ADR(ErrorLog));
		END_CASE;

	(* ******************************************************************************************************** *)
	(* Manual *)
	(* ******************************************************************************************************** *)
	CmdMAN:
		CASE CmdExe.CmdCase OF
			(* Case 0 *)
			0: 	TFStateUpdate(ADR(State),StateMAN_RUN);
				TFTimerSet(ADR(Timeout),10,TRUE);
				IF TFCommandParRead(CmdExe.Cmd.Parameter,ADR(ParametersArray),2) THEN
					MAN_Actuator	:= STRING_TO_UINT(ParametersArray.Parameters[0]);
					MAN_Cmd		:= STRING_TO_UINT(ParametersArray.Parameters[1]);
				ELSE
					TFError(ErrCMDPARNUM,ErrNULL,ADR(CmdExe),ADR(State),ADR(Error),ADR(ErrorLog));
					RETURN;
				END_IF;

				CASE MAN_Actuator OF
					(* Case 0..99 for Actuators *)
					(* Case 100..199  for Axis *)

					(* Case Nop *)
					0:	;

					(* Case 1: *)
					1:	CASE MAN_Cmd OF
							0:	;
							
							(* Case 10: Suction OFF *)
							10:	OUT.EV_Suction := FALSE;
								
							(* Case 11: Suction ON *)
							11:	OUT.EV_Suction := TRUE;

							(* Case 10: Suction Cup Up *)
							20:	OUT.EV_SuctionCupsUp := TRUE;
								OUT.EV_SuctionCupsDown := FALSE;

							(* Case 11: Suction Cup Down *)
							21:	OUT.EV_SuctionCupsUp := FALSE;
								OUT.EV_SuctionCupsDown := TRUE;

							ELSE
								TFError(ErrNOCMDCASE,ErrNULL,ADR(CmdExe),ADR(State),ADR(Error),ADR(ErrorLog));
						END_CASE;

					100:CASE MAN_Cmd OF
							0:	;
							ELSE
								TFError(ErrNOCMDCASE,ErrNULL,ADR(CmdExe),ADR(State),ADR(Error),ADR(ErrorLog));
						END_CASE;

					ELSE
						TFError(ErrNOCMDCASE,ErrNULL,ADR(CmdExe),ADR(State),ADR(Error),ADR(ErrorLog));
				END_CASE;

				IF CmdExe.CmdCase = 0 THEN
					TFCommandCase(ADR(CmdExe),1,CommandCase_INC);
				END_IF

			(* Case 1 *)
			1: 	IF (MAN_Cmd = 0) OR TFTimerDone(ADR(Timeout)) THEN
					(* Clear All Output Here *)
					;
					TFStateUpdate(ADR(State),StateMAN_END);
					TFCommandExeClear(ADR(CmdExe));
				END_IF;
			10: ;
			(* Case 100 - End *)
			100:(* Clear All Output Here *)
				TFStateUpdate(ADR(State),StateMAN_END);
				TFCommandExeClear(ADR(CmdExe));

			ELSE
				TFError(ErrNOCMDCASE,ErrNULL,ADR(CmdExe),ADR(State),ADR(Error),ADR(ErrorLog));
		END_CASE;

	(* ******************************************************************************************************** *)
	(* LOAD - Attivazione aspirazione + discesa ventose *)
	(* ******************************************************************************************************** *)
		CmdLOAD:
		CASE CmdExe.CmdCase OF
			
			(* Case 0 - Init Command*)
			0: 	TFStateUpdate(ADR(State),StateLoad_RUN);
				TFTimerSet(ADR(Timeout),60000,TRUE);
				TFCommandCase(ADR(CmdExe),1,CommandCase_INC);
				
			(* Case 1 - Attivazione Ventosa *)					
			1:
				OUT.EV_Suction := TRUE;
				TFCommandCase(ADR(CmdExe),1,CommandCase_INC);
			(* Case 2 - Discesa Ventose *)		
			2: 
				OUT.EV_SuctionCupsDOWN 	:= TRUE;
				OUT.EV_SuctionCupsUP 	:= FALSE;
				TFTimerSet(ADR(TimerAspirazione),2000,TRUE);
				TFCommandCase(ADR(CmdExe),1,CommandCase_INC);
			3:
				IF TFTimerDone(ADR(TimerAspirazione)) THEN
					TFCommandCase(ADR(CmdExe),100,CommandCase_JMP);
				END_IF
				
			(* Case 100 *)
			100:TFStateUpdate(ADR(State),StateLOAD_END);
				TFCommandExeClear(ADR(CmdExe));

			ELSE
				TFError(ErrNOCMDCASE,ErrNULL,ADR(CmdExe),ADR(State),ADR(Error),ADR(ErrorLog));
		END_CASE
		
	(* ******************************************************************************************************** *)
	(* UNLOAD - Attivazione aspirazione + discesa ventose *)
	(* ******************************************************************************************************** *)
		CmdUNLOAD:
		CASE CmdExe.CmdCase OF
			
			(* Case 0 - Init Command*)
			0: 	TFStateUpdate(ADR(State),StateUNLOAD_RUN);
				TFTimerSet(ADR(Timeout),60000,TRUE);
				TFCommandCase(ADR(CmdExe),1,CommandCase_INC);
				
			(* Case 1 - Disattivazione Aspirazione*)					
			1:	
				OUT.EV_Suction := False;
				TFCommandCase(ADR(CmdExe),1,CommandCase_INC);
			
			(* Case 2 - Salita Ventose *)		
			2: 
				OUT.EV_SuctionCupsDOWN 	:= FALSE;
				OUT.EV_SuctionCupsUP 	:= TRUE;
				TFCommandCase(ADR(CmdExe),100,CommandCase_JMP);	
				
			(* Case 100 *)
			100:TFStateUpdate(ADR(State),StateUNLOAD_END);
				TFCommandExeClear(ADR(CmdExe));

			ELSE
				TFError(ErrNOCMDCASE,ErrNULL,ADR(CmdExe),ADR(State),ADR(Error),ADR(ErrorLog));
		END_CASE
	ELSE
		TFError(ErrNOCMD,ErrNULL,ADR(CmdExe),ADR(State),ADR(Error),ADR(ErrorLog));

END_CASE;


(* ******************************************************************************************************** *)
(* State Input/Output *)
(* ******************************************************************************************************** *)
(* Fill Input/Output bit with sensor, electrovalve, etc. status *)


(* ******************************************************************************************************** *)
(* Input *)
(* ******************************************************************************************************** *)

(* ******************************************************************************************************** *)
(* Alarm *)
(* ******************************************************************************************************** *)

(* ******************************************************************************************************** *)
(* Error Check - Clear All Output!!! *)
(* ******************************************************************************************************** *)
IF Error.Code > ErrNULL THEN
	IF CmdExe.Code <> CmdNOP THEN
		IF CmdExe.Code <> CmdSTOP AND
			CmdExe.Code <> CmdPOWER AND
			CmdExe.Code <> CmdRESET AND
			CmdExe.Code <> CmdMAN AND
			CmdExe.Code <> CmdLOAD AND
			CmdExe.Code <> CmdUNLOAD THEN
			TFCommandClear(ADR(CmdNext));
			TFCommandExeClear(ADR(CmdExe));

			(* Clear All Output Here *)

		END_IF;
	END_IF;
END_IF;


(* ******************************************************************************************************** *)
(* Common Outputs *)
(* ******************************************************************************************************** *)

END_FUNCTION_BLOCK

// ---- Data types/AlbertoPruevas/BloqueFunciones/Fb_SensoresTasteggio.TcPOU
FUNCTION_BLOCK Fb_SensoresTasteggio
VAR_INPUT
	Sensor_Tasteo_1 				: BOOL ;
	Sensor_Tasteo_2 				: BOOL ;
	Sensor_Tasteo_3 				: BOOL ;
	Sensor_Tasteo_4 				: BOOL ;
	Nu_sensores_Dar_Out				: BYTE ;
END_VAR
VAR_OUTPUT
	Sensores_Tasteggio_Ok 			: BOOL ;
	Nu_Sesores_Activos				: BYTE ;
END_VAR
VAR
END_VAR

Nu_Sesores_Activos := BOOL_TO_BYTE(Sensor_Tasteo_1) + BOOL_TO_BYTE(Sensor_Tasteo_2) + BOOL_TO_BYTE(Sensor_Tasteo_3) + BOOL_TO_BYTE(Sensor_Tasteo_4) ; 

IF Nu_Sesores_Activos >= Nu_sensores_Dar_Out THEN
	Sensores_Tasteggio_Ok := TRUE ;
	ELSE
	Sensores_Tasteggio_Ok := FALSE ;	
	
END_IF

END_FUNCTION_BLOCK

// ---- Data types/AlbertoPruevas/Funciones/FuncionesFormaciones/Fun_CalculoCoordenadasFinalesFormacion.TcPOU
FUNCTION Fun_CalculoCoordenadasFinalesFormacion : bool
VAR_INPUT
	TipoCalForCavallete 		: UINT ;
	numeroLastre_int 		: UINT ;
	Supporto 				: POINTER TO TFMachinePalletizer_Pallet;
	XFinale 				: POINTER TO  ARRAY [1..MAXFORMINGSLAB] OF LREAL;
	YFinale 				: POINTER TO  ARRAY [1..MAXFORMINGSLAB] OF LREAL;
	YInternoLastra 			: POINTER TO  ARRAY [1..MAXFORMINGSLAB] OF LREAL;
	ZFinale 				: POINTER TO  ARRAY [1..MAXFORMINGSLAB] OF LREAL;
	ZInternoLastra			: POINTER TO  ARRAY [1..MAXFORMINGSLAB] OF LREAL;
	JFinale 				: POINTER TO  ARRAY [1..MAXFORMINGSLAB] OF LREAL;
END_VAR
VAR
	Contador: UINT;
END_VAR

FOR Contador := 1 TO numeroLastre_int * 2 DO 
	CASE TipoCalForCavallete OF 
		1: 

			XFinale^[Contador] := Supporto^.XDim/2 + Supporto^.OFSDE_X180;
			;
		2: 
			;
		3:
			;
		4: 
			;
	END_CASE
	
END_FOR

END_FUNCTION

// ---- POUs/Check/CheckBounds.TcPOU
// Implicitly generated code : DO NOT EDIT
FUNCTION CheckBounds : DINT
VAR_INPUT
	index, lower, upper: DINT;
END_VAR

// Implicitly generated code : Only an Implementation suggestion
{noflow}
IF  index < lower THEN
	CheckBounds := lower;
ELSIF  index > upper THEN
	CheckBounds := upper;
ELSE  
	CheckBounds := index;
END_IF
{flow}

END_FUNCTION

// ---- POUs/Check/CheckDivDInt.TcPOU
// Implicitly generated code : DO NOT EDIT
FUNCTION CheckDivDInt : DINT
VAR_INPUT
	divisor:DINT;
END_VAR

// Implicitly generated code : Only an Implementation suggestion
{noflow}
IF divisor = 0 THEN
	CheckDivDInt:=1;
ELSE
	CheckDivDInt:=divisor;
END_IF;
{flow}

END_FUNCTION

// ---- POUs/Check/CheckDivLInt.TcPOU
// Implicitly generated code : DO NOT EDIT
FUNCTION CheckDivLInt : LINT
VAR_INPUT
	divisor:LINT;
END_VAR

// Implicitly generated code : Only an Implementation suggestion
{noflow}
IF divisor = 0 THEN
	CheckDivLInt:=1;
ELSE
	CheckDivLInt:=divisor;
END_IF;
{flow}

END_FUNCTION

// ---- POUs/Check/CheckDivLReal.TcPOU
// Implicitly generated code : DO NOT EDIT
FUNCTION CheckDivLReal : LREAL
VAR_INPUT
	divisor:LREAL;
END_VAR

// Implicitly generated code : Only an Implementation suggestion
{noflow}
IF divisor = 0 THEN
	CheckDivLReal:=1;
ELSE
	CheckDivLReal:=divisor;
END_IF;
{flow}

END_FUNCTION

// ---- POUs/Check/CheckDivReal.TcPOU
// Implicitly generated code : DO NOT EDIT
FUNCTION CheckDivReal : REAL
VAR_INPUT
	divisor:REAL;
END_VAR

// Implicitly generated code : Only an Implementation suggestion
{noflow}
IF divisor = 0 THEN
	CheckDivReal:=1;
ELSE
	CheckDivReal:=divisor;
END_IF;
{flow}

END_FUNCTION

// ---- POUs/Check/CheckLRangeSigned.TcPOU
// Implicitly generated code : DO NOT EDIT
FUNCTION CheckLRangeSigned : LINT
VAR_INPUT
	value, lower, upper: LINT;
END_VAR

// Implicitly generated code : Only an Implementation suggestion
{noflow}
IF (value < lower) THEN
	CheckLRangeSigned := lower;
ELSIF(value > upper) THEN
	CheckLRangeSigned := upper;
ELSE
	CheckLRangeSigned := value;
END_IF

{flow}

END_FUNCTION

// ---- POUs/Check/CheckLRangeUnsigned.TcPOU
// Implicitly generated code : DO NOT EDIT
FUNCTION CheckLRangeUnsigned : ULINT
VAR_INPUT
	value, lower, upper: ULINT;
END_VAR

// Implicitly generated code : Only an Implementation suggestion
{noflow}
IF (value < lower) THEN
	CheckLRangeUnsigned := lower;
ELSIF(value > upper) THEN
	CheckLRangeUnsigned := upper;
ELSE
	CheckLRangeUnsigned := value;
END_IF
{flow}

END_FUNCTION

// ---- POUs/Check/CheckPointer.TcPOU
// Implicitly generated code : DO NOT EDIT
FUNCTION CheckPointer : POINTER TO BYTE
VAR_INPUT 
	ptToTest : POINTER TO BYTE; // Destination address of the pointer
	iSize : DINT;		        // Size of the type the pointer points to. (e.g: 20 for POINTER TO ARRAY [0..9] OF INT) 
	iGran : DINT;		        // Granularity of the pointer access. This is the size of the biggest non-structured data type in the type the pointer points to. (e.g: 2 for POINTER TO ARRAY [0..9] OF INT)
	bWrite: BOOL;		        // Indicates read or write Access. TRUE = write access.
END_VAR

// Implicitly generated code : Only an Implementation suggestion
{noflow}
IF NOT FirstStatrtEx THEN
IF ptToTest=0 THEN
    ADSLOGSTR(ADSLOG_MSGTYPE_ERROR OR ADSLOG_MSGTYPE_STRING,'CheckPointer failed due to invalid address.','');
ELSIF iSize<=0 THEN
    ADSLOGSTR(ADSLOG_MSGTYPE_ERROR OR ADSLOG_MSGTYPE_STRING,'CheckPointer failed due to invalid size.','');
ELSIF iGran<=0 THEN
    ADSLOGSTR(ADSLOG_MSGTYPE_ERROR OR ADSLOG_MSGTYPE_STRING,'CheckPointer failed due to invalid granularity.','');
// -> Please note that the following memory area check is time consuming:
//ELSIF F_CheckMemoryArea(pData:=ptToTest,nSize:=DINT_TO_UDINT(iSize)) = E_TcMemoryArea.Unknown THEN
//    ADSLOGSTR(ADSLOG_MSGTYPE_ERROR OR ADSLOG_MSGTYPE_STRING,'CheckPointer failed due to unknown memory area.','');
END_IF
CheckPointer := ptToTest;
END_IF
{flow}

END_FUNCTION

// ---- POUs/Check/CheckRangeSigned.TcPOU
// Implicitly generated code : DO NOT EDIT
FUNCTION CheckRangeSigned : DINT
VAR_INPUT
	value, lower, upper: DINT;
END_VAR

// Implicitly generated code : Only an Implementation suggestion
{noflow}
IF (value < lower) THEN
	CheckRangeSigned := lower;
ELSIF(value > upper) THEN
	CheckRangeSigned := upper;
ELSE
	CheckRangeSigned := value;
END_IF
{flow}

END_FUNCTION

// ---- POUs/Check/CheckRangeUnsigned.TcPOU
// Implicitly generated code : DO NOT EDIT
FUNCTION CheckRangeUnsigned : UDINT
VAR_INPUT
	value, lower, upper: UDINT;
END_VAR

// Implicitly generated code : Only an Implementation suggestion
{noflow}
IF (value < lower) THEN
	CheckRangeUnsigned := lower;
ELSIF(value > upper) THEN
	CheckRangeUnsigned := upper;
ELSE
	CheckRangeUnsigned := value;
END_IF
{flow}

END_FUNCTION

// ---- POUs/TFGateAccess/TFGateAccess.TcPOU
FUNCTION_BLOCK TFGateAccess
VAR_INPUT
	MachineCmd : POINTER TO CommandBuffer;
	MachineCmdExe : POINTER TO CommandExe;
	MachineState : POINTER TO State;
	MachineError : POINTER TO Error;
	MachineMode : POINTER TO Mode;
	
	TimeBase : REAL;
	AccessRequest : BOOL;
	AccessDone : BOOL;
	LGVAccessActive	: BOOL;
	TilterPhaseStopDone : BOOL;
	PowerOK : BOOL;//Indica la presenza della marcia
	DisableStopEpowerOFF : BOOL;
END_VAR
VAR_OUTPUT
	AccessLamp : BOOL; (* Access Lamp: 	OFF = No Access Consent,
										ON = Access Consent,
										FLASH (1sec) = Access Requested (Machine Stopping)
										FLASH (0.5sec) = Waiting Restart
										FLASH (0.1sec) = Access Error *)
										
	AccesActive : BOOL; (* Gate Acces Sequence in Execution *)
	AccessOK : BOOL;	(* Accesso consentito *)
	TilterPhaseStop : BOOL;		
	AccessERRORCode : UINT;		
	ErrAck : BOOL;
	ErrAckDriver : BOOL;			
END_VAR
VAR
	ParametersArray : ParametersArray;
	
	AccessERROR : BOOL;
	AccessReqIN : BOOL;
	AccessReqOUT : BOOL;
	AccessCase : INT;
	MachineWasRunning : BOOL;
	MachineWasRunning2 : bool;
	Timer100 : REAL;
	Timer500 : REAL;
	Timer1000 : REAL;
	Clock100 : BOOL;
	Clock500 : BOOL;
	Clock1000 : BOOL;
	TimerPowerOFF : real;
	MEMDiMarciaInPartenza : BOOL;
	TimerRitardoPower : REAL;
END_VAR

TFTimerCall(ADR(Timer100),TimeBase);
TFTimerCall(ADR(Timer500),TimeBase);
TFTimerCall(ADR(Timer1000),TimeBase);
TFTimerCall(ADR(TimerPowerOFF),TimeBase);
TFTimerCall(ADR(TimerRitardoPower),TimeBase);

CASE AccessCase OF
	
	(* Wait Request ON *)
	0:	AccesActive := FALSE;
		AccessOK := FALSE;
		AccessReqIN := FALSE;
		AccessReqOUT := FALSE;
		
		IF AccessRequest AND NOT AccessDone (*AND NOT LGVAccessActive*) AND NOT TFIsModuleError(MachineError^) THEN
			AccesActive := TRUE;
			AccessERROR := FALSE;
			AccessReqIN := TRUE;
			(* Machine Was Running if CmdDO and No Stop Request *) 
			MachineWasRunning := MachineCmdExe^.Code = CmdDO AND MachineCmdExe^.PhaseStopRequest = 0 AND MachineCmdExe^.RapidStopRequest = 0;
			IF NOT DisableStopEpowerOFF THEN
				AccessCase := 10;
			ELSE
				AccessCase := 10;
			END_IF
		ELSIF AccessERROR THEN
			AccessERRORCode := 0;
			AccessERROR := FALSE;
			TilterPhaseStop := false;
		END_IF
		
	(* Phase Stop *)
	10:	TFParametersArrayClear(ADR(ParametersArray));
		TFCommandSend(CmdSTOPPHASE,ParametersArray,MachineCmd^);
		AccessCase := AccessCase + 1;
		
	11:	IF ((TFStateCodeGet(MachineState^) = StateDO_END OR
			MachineCmdExe^.Code = CmdNOP)) THEN
				TFTimerSet(ADR(TimerPowerOFF),100,TRUE);
				AccessCase := 20;
		ELSIF TFIsModuleError(MachineError^) THEN
			AccessERRORCode := ErrMACHINEPALLETIZER_ERRORE_MACCHINA_IN_RICHIN;
			TilterPhaseStop := TRUE;
			AccessERROR := TRUE;
			AccessCase := 0;
		END_IF

	(* Power Off *)
	20:	//Valuto se nel pal è presente la marcia, in questo modo alla fine della rich. di ingresso do o meno il power
		IF PowerOK THEN
			MEMDiMarciaInPartenza := TRUE;
		ELSE
			MEMDiMarciaInPartenza := FALSE;
		END_IF
		IF TFTimerDone(ADR(TimerPowerOFF)) THEN
			TilterPhaseStop := FALSE;
			TFParametersArrayClear(ADR(ParametersArray));
			ParametersArray.Parameters[0] := '0';
			TFCommandSend(CmdPOWER,ParametersArray,MachineCmd^);
			AccessCase := AccessCase + 1;
		ELSIF TFIsModuleError(MachineError^) THEN
			AccessERRORCode := ErrMACHINEPALLETIZER_ERRORE_MACCHINA_IN_RICHIN;
			AccessERROR := TRUE;
			AccessCase := 0;
		ELSIF NOT AccessRequest THEN
			TilterPhaseStop := FALSE;
			AccessCase := 0;
		END_IF	

	21:	IF TFStateCodeGet(MachineState^) = StatePOWER_END THEN
			AccessCase := 25;
		ELSIF TFIsModuleError(MachineError^) THEN
			AccessERRORCode := ErrMACHINEPALLETIZER_ERRORE_MACCHINA_IN_RICHIN;
			AccessERROR := TRUE;
			AccessCase := 0;
		END_IF
		
	25:(* Access Ok.... Wait Request Done ON *)
		AccessReqIN := FALSE;
		AccessReqOUT := FALSE;
		AccessOK := TRUE;
		IF NOT AccessRequest AND AccessDone THEN
			AccessCase := AccessCase + 1;
			TFTimerSet(ADR(TimerRitardoPower),100,TRUE);
			ErrAck := TRUE;
		END_IF
		IF TFIsModuleError(MachineError^) THEN
			AccessERRORCode := ErrMACHINEPALLETIZER_ERRORE_MACCHINA_IN_RICHIN;
			AccessERROR := TRUE;
			AccessCase := 0;
		END_IF
		
	26:
		IF TFTimerDone(ADR(TimerRitardoPower)) THEN
			TFTimerSet(ADR(TimerRitardoPower),100,TRUE);
			ErrAck := FALSE;
			AccessCase := 27;
		END_IF
		
	27:
		IF TFTimerDone(ADR(TimerRitardoPower)) THEN
			TFTimerSet(ADR(TimerRitardoPower),100,TRUE);
			ErrAckDriver := TRUE;
			AccessCase := 30;
		END_IF

	(* Access Ok.... Wait Request Done ON *)
	30:	//AccessReqIN := FALSE;
		//AccessReqOUT := FALSE;
		//AccessOK := TRUE;
		//IF NOT AccessRequest AND AccessDone THEN
		IF TFTimerDone(ADR(TimerRitardoPower)) THEN
			AccessCase := 31;
			TFTimerSet(ADR(TimerRitardoPower),100,TRUE);
			ErrAckDriver := FALSE;
		END_IF
		//END_IF
		IF TFIsModuleError(MachineError^) THEN
			AccessERRORCode := ErrMACHINEPALLETIZER_ERRORE_MACCHINA_IN_RICHIN;
			AccessERROR := TRUE;
			AccessCase := 0;
		END_IF

	(* Wait Request Done OFF *)
	31:	TFTimerSet(ADR(TimerRitardoPower),100,AccessDone);
		IF NOT AccessDone AND TFTimerDone(ADR(TimerRitardoPower))THEN
			AccessOK := FALSE;
			AccessReqOUT := TRUE;
			AccessCase := 40;
			ErrAckDriver := FALSE;
		ELSIF TFIsModuleError(MachineError^) THEN
			AccessERRORCode := ErrMACHINEPALLETIZER_ERRORE_MACCHINA_IN_RICHIN;
			AccessERROR := TRUE;
			AccessCase := 0;
		END_IF
		
	(* Power ON *)
	40:	IF NOT LGVAccessActive THEN
			IF MEMDiMarciaInPartenza THEN
				TFParametersArrayClear(ADR(ParametersArray));
				ParametersArray.Parameters[0] := '1';
				TFCommandSend(CmdPOWER,ParametersArray,MachineCmd^);
				AccessCase := AccessCase + 1;
			ELSE
				AccessCase := 50;
			END_IF		
		ELSE
			AccessCase := 50;
		END_IF	

	41:	IF TFStateCodeGet(MachineState^) = StatePOWER_END THEN //OR TFIsModuleError(MachineError^) THEN
			AccessCase := 50;
		ELSIF TFIsModuleError(MachineError^) THEN
			AccessERRORCode := ErrMACHINEPALLETIZER_ERRORE_MACCHINA_IN_RICHIN;
			AccessERROR := TRUE;
			AccessCase := 0;
		END_IF

	50:	IF NOT AccessRequest AND AccessDone THEN
			AccessCase := AccessCase + 1;
		END_IF

	(* Wait Request Done OFF *)
	51:	IF NOT AccessDone THEN
			AccessCase := 60;
		END_IF

	(* Machine Restart *)
	60:	AccessCase := AccessCase + 1;
		IF MachineWasRunning AND
			MachineMode^.Auto AND
			NOT MachineMode^.StopRequest AND
			NOT MachineMode^.RapidStopRequest AND NOT LGVAccessActive THEN
				TFParametersArrayClear(ADR(ParametersArray));
				TFCommandSend(CmdDO,ParametersArray,MachineCmd^);		
		ELSIF TFIsModuleError(MachineError^) THEN
			AccessERRORCode := ErrMACHINEPALLETIZER_ERRORE_MACCHINA_IN_RICHIN;
			AccessERROR := TRUE;
			AccessCase := 0;
		END_IF
			
	61:	AccessReqIN := FALSE;
		AccessReqOUT := FALSE;
		AccessOK := FALSE;
		AccessCase := 0;
		MEMDiMarciaInPartenza := FALSE;
		
		
	//80:
	//	AccessOK := FALSE;
	//	IF NOT AccessRequest AND AccessDone THEN
	//		AccessCase := AccessCase + 1;
	//	END_IF
		
	ELSE
		AccessERROR := TRUE;
		AccessERRORCode := ErrMACHINEPALLETIZER_ERRORE_MACCHINA_IN_RICHIN;
		MEMDiMarciaInPartenza := FALSE;
		AccessCase := 0;
		
END_CASE

(* Clocks *)
IF TFTimerDone(ADR(Timer100)) THEN
	TFTimerSet(ADR(Timer100),100,TRUE);
	Clock100 := NOT Clock100;
END_IF
IF TFTimerDone(ADR(Timer500)) THEN
	TFTimerSet(ADR(Timer500),500,TRUE);
	Clock500 := NOT Clock500;
END_IF
IF TFTimerDone(ADR(Timer1000)) THEN
	TFTimerSet(ADR(Timer1000),1000,TRUE);
	Clock1000 := NOT Clock1000;
END_IF

(* Access Lamp *)
AccessLamp := 	(AccessOK OR
				(AccessReqOUT AND Clock500) OR
				(AccessReqIN AND Clock1000))AND
				NOT AccessERROR OR (AccessERROR AND Clock100);

END_FUNCTION_BLOCK

// ---- POUs/TFGateAccess/TFGateAccessDoppiaMacchina.TcPOU
(* Copyright (c) 2015 Fausto Bellei - fbellei@creoevolution.com - CREO EVOLUTION SRL - http://www.creoevolution.com *)

(* Permission is hereby granted, free of charge, to any person obtaining a copy of this software and associated documentation files (the "Software"), to deal in the
   Software without restriction, including without limitation the rights to use, copy, modify, merge, publish, distribute, sublicense, and/or sell copies of the Software,
   and to permit persons to whom the Software is furnished to do so, subject to the following conditions:

   The above copyright notice and this permission notice shall be included in all copies or substantial portions of the Software.

   THE SOFTWARE IS PROVIDED "AS IS", WITHOUT WARRANTY OF ANY KIND, EXPRESS OR IMPLIED, INCLUDING BUT NOT LIMITED TO THE WARRANTIES OF
   MERCHANTABILITY, FITNESS FOR A PARTICULAR PURPOSE AND NONINFRINGEMENT. IN NO EVENT SHALL THE AUTHORS OR COPYRIGHT HOLDERS BE LIABLE FOR
   ANY CLAIM, DAMAGES OR OTHER LIABILITY, WHETHER IN AN ACTION OF CONTRACT, TORT OR OTHERWISE, ARISING FROM, OUT OF OR IN CONNECTION WITH THE
   SOFTWARE OR THE USE OR OTHER DEALINGS IN THE SOFTWARE. *)

FUNCTION_BLOCK TFGateAccessDoppiaMacchina
VAR_INPUT
	MachineCmd : POINTER TO CommandBuffer;
	MachineCmdExe : POINTER TO CommandExe;
	MachineState : POINTER TO State;
	MachineError : POINTER TO Error;
	MachineMode : POINTER TO Mode;
	
	MachineCmd2 : POINTER TO CommandBuffer;//Macchina 2
	MachineCmdExe2 : POINTER TO CommandExe;//Macchina 2
	MachineState2 : POINTER TO State;//Macchina 2
	MachineError2 : POINTER TO Error;//Macchina 2
	MachineMode2 : POINTER TO Mode;//Macchina 2

	TimeBase : REAL;
	AccessRequest : BOOL;
	AccessDone : BOOL;
	LGVAccessActive	: BOOL;
	TilterPhaseStopDone : BOOL;
	PowerOK : BOOL;//Indica la presenza della marcia
END_VAR
VAR_OUTPUT
	AccessLamp : BOOL; (* Access Lamp: 	OFF = No Access Consent,
										ON = Access Consent,
										FLASH (1sec) = Access Requested (Machine Stopping)
										FLASH (0.5sec) = Waiting Restart
										FLASH (0.1sec) = Access Error *)
										
	AccesActive : BOOL; (* Gate Acces Sequence in Execution *)
	AccessOK : BOOL;	(* Accesso consentito *)
	TilterPhaseStop : BOOL;		
	AccessERRORCode : UINT;		
	ErrAck : BOOL;
	ErrAckDriver : BOOL;			
END_VAR
VAR
	ParametersArray : ParametersArray;
	
	AccessERROR : BOOL;
	AccessReqIN : BOOL;
	AccessReqOUT : BOOL;
	AccessCase : INT;
	MachineWasRunning : BOOL;
	MachineWasRunning2 : bool;
	Timer100 : REAL;
	Timer500 : REAL;
	Timer1000 : REAL;
	Clock100 : BOOL;
	Clock500 : BOOL;
	Clock1000 : BOOL;
	TimerPowerOFF : real;
	MEMDiMarciaInPartenza : BOOL;
	TimerRitardoPower : REAL;
END_VAR

TFTimerCall(ADR(Timer100),TimeBase);
TFTimerCall(ADR(Timer500),TimeBase);
TFTimerCall(ADR(Timer1000),TimeBase);
TFTimerCall(ADR(TimerPowerOFF),TimeBase);
TFTimerCall(ADR(TimerRitardoPower),TimeBase);

CASE AccessCase OF
	
	(* Wait Request ON *)
	0:	AccesActive := FALSE;
		AccessOK := FALSE;
		AccessReqIN := FALSE;
		AccessReqOUT := FALSE;
		
		IF AccessRequest AND NOT AccessDone (*AND NOT LGVAccessActive*) AND NOT TFIsModuleError(MachineError^) AND NOT TFIsModuleError(MachineError2^) THEN
			AccesActive := TRUE;
			AccessERROR := FALSE;
			AccessReqIN := TRUE;
			(* Machine Was Running if CmdDO and No Stop Request *) 
			MachineWasRunning := MachineCmdExe^.Code = CmdDO AND MachineCmdExe^.PhaseStopRequest = 0 AND MachineCmdExe^.RapidStopRequest = 0;
			MachineWasRunning2 := MachineCmdExe2^.Code = CmdDO AND MachineCmdExe2^.PhaseStopRequest = 0 AND MachineCmdExe2^.RapidStopRequest = 0;
			AccessCase := 10;
		ELSIF AccessERROR THEN
			AccessERRORCode := 0;
			AccessERROR := FALSE;
			TilterPhaseStop := false;
		END_IF
		
	(* Phase Stop *)
	10:	TFParametersArrayClear(ADR(ParametersArray));
		TFCommandSend(CmdSTOPPHASE,ParametersArray,MachineCmd^);
		TFCommandSend(CmdSTOPPHASE,ParametersArray,MachineCmd2^);
		AccessCase := AccessCase + 1;
		
	11:	IF ((TFStateCodeGet(MachineState^) = StateDO_END OR
			MachineCmdExe^.Code = CmdNOP)) AND
			((TFStateCodeGet(MachineState2^) = StateDO_END OR
			MachineCmdExe2^.Code = CmdNOP)) THEN
				TFTimerSet(ADR(TimerPowerOFF),100,TRUE);
				AccessCase := 20;
		ELSIF TFIsModuleError(MachineError^) OR TFIsModuleError(MachineError2^) THEN
			AccessERRORCode := ErrMACHINEPALLETIZER_ERRORE_MACCHINA_IN_RICHIN;
			TilterPhaseStop := TRUE;
			AccessERROR := TRUE;
			AccessCase := 0;
		END_IF

	(* Power Off *)
	20:	//Valuto se nel pal è presente la marcia, in questo modo alla fine della rich. di ingresso do o meno il power
		IF PowerOK THEN
			MEMDiMarciaInPartenza := TRUE;
		ELSE
			MEMDiMarciaInPartenza := FALSE;
		END_IF
		IF TFTimerDone(ADR(TimerPowerOFF)) THEN
			TilterPhaseStop := FALSE;
			TFParametersArrayClear(ADR(ParametersArray));
			ParametersArray.Parameters[0] := '0';
			TFCommandSend(CmdPOWER,ParametersArray,MachineCmd^);
			TFCommandSend(CmdPOWER,ParametersArray,MachineCmd2^);
			AccessCase := AccessCase + 1;
		ELSIF TFIsModuleError(MachineError^) OR  TFIsModuleError(MachineError2^) THEN
			AccessERRORCode := ErrMACHINEPALLETIZER_ERRORE_MACCHINA_IN_RICHIN;
			AccessERROR := TRUE;
			AccessCase := 0;
		ELSIF NOT AccessRequest THEN
			TilterPhaseStop := FALSE;
			AccessCase := 0;
		END_IF	

	21:	IF TFStateCodeGet(MachineState^) = StatePOWER_END AND TFStateCodeGet(MachineState2^) = StatePOWER_END THEN
			AccessCase := 25;
		ELSIF TFIsModuleError(MachineError^) OR TFIsModuleError(MachineError2^) THEN
			AccessERRORCode := ErrMACHINEPALLETIZER_ERRORE_MACCHINA_IN_RICHIN;
			AccessERROR := TRUE;
			AccessCase := 0;
		END_IF
		
	25:(* Access Ok.... Wait Request Done ON *)
		AccessReqIN := FALSE;
		AccessReqOUT := FALSE;
		AccessOK := TRUE;
		IF NOT AccessRequest AND AccessDone THEN
			AccessCase := AccessCase + 1;
			TFTimerSet(ADR(TimerRitardoPower),100,TRUE);
			ErrAck := TRUE;
		END_IF
		IF TFIsModuleError(MachineError^) OR TFIsModuleError(MachineError2^) THEN
			AccessERRORCode := ErrMACHINEPALLETIZER_ERRORE_MACCHINA_IN_RICHIN;
			AccessERROR := TRUE;
			AccessCase := 0;
		END_IF
		
	26:
		IF TFTimerDone(ADR(TimerRitardoPower)) THEN
			TFTimerSet(ADR(TimerRitardoPower),100,TRUE);
			ErrAck := FALSE;
			AccessCase := 27;
		END_IF
		
	27:
		IF TFTimerDone(ADR(TimerRitardoPower)) THEN
			TFTimerSet(ADR(TimerRitardoPower),100,TRUE);
			ErrAckDriver := TRUE;
			AccessCase := 30;
		END_IF

	(* Access Ok.... Wait Request Done ON *)
	30:	//AccessReqIN := FALSE;
		//AccessReqOUT := FALSE;
		//AccessOK := TRUE;
		//IF NOT AccessRequest AND AccessDone THEN
		IF TFTimerDone(ADR(TimerRitardoPower)) THEN
			AccessCase := 31;
			TFTimerSet(ADR(TimerRitardoPower),100,TRUE);
			ErrAckDriver := FALSE;
		END_IF
		//END_IF
		IF TFIsModuleError(MachineError^) OR TFIsModuleError(MachineError2^) THEN
			AccessERRORCode := ErrMACHINEPALLETIZER_ERRORE_MACCHINA_IN_RICHIN;
			AccessERROR := TRUE;
			AccessCase := 0;
		END_IF

	(* Wait Request Done OFF *)
	31:	TFTimerSet(ADR(TimerRitardoPower),100,AccessDone);
		IF NOT AccessDone AND TFTimerDone(ADR(TimerRitardoPower))THEN
			AccessOK := FALSE;
			AccessReqOUT := TRUE;
			AccessCase := 40;
			ErrAckDriver := FALSE;
		ELSIF TFIsModuleError(MachineError^) OR TFIsModuleError(MachineError2^) THEN
			AccessERRORCode := ErrMACHINEPALLETIZER_ERRORE_MACCHINA_IN_RICHIN;
			AccessERROR := TRUE;
			AccessCase := 0;
		END_IF
		
	(* Power ON *)
	40:	IF NOT LGVAccessActive THEN
			IF MEMDiMarciaInPartenza THEN
				TFParametersArrayClear(ADR(ParametersArray));
				ParametersArray.Parameters[0] := '1';
				TFCommandSend(CmdPOWER,ParametersArray,MachineCmd^);
				TFCommandSend(CmdPOWER,ParametersArray,MachineCmd2^);
				AccessCase := AccessCase + 1;
			ELSE
				AccessCase := 50;
			END_IF		
		ELSE
			AccessCase := 50;
		END_IF	

	41:	IF TFStateCodeGet(MachineState^) = StatePOWER_END AND  TFStateCodeGet(MachineState2^) = StatePOWER_END THEN //OR TFIsModuleError(MachineError^) THEN
			AccessCase := 50;
		ELSIF TFIsModuleError(MachineError^) OR TFIsModuleError(MachineError2^) THEN
			AccessERRORCode := ErrMACHINEPALLETIZER_ERRORE_MACCHINA_IN_RICHIN;
			AccessERROR := TRUE;
			AccessCase := 0;
		END_IF

	50:	IF NOT AccessRequest AND AccessDone THEN
			AccessCase := AccessCase + 1;
		END_IF

	(* Wait Request Done OFF *)
	51:	IF NOT AccessDone THEN
			AccessCase := 60;
		END_IF

	(* Machine Restart *)
	60:	AccessCase := AccessCase + 1;
		IF MachineWasRunning AND
			MachineMode^.Auto AND
			NOT MachineMode^.StopRequest AND
			NOT MachineMode^.RapidStopRequest AND NOT LGVAccessActive THEN
				TFParametersArrayClear(ADR(ParametersArray));
				TFCommandSend(CmdDO,ParametersArray,MachineCmd^);		
		ELSIF TFIsModuleError(MachineError^) THEN
			AccessERRORCode := ErrMACHINEPALLETIZER_ERRORE_MACCHINA_IN_RICHIN;
			AccessERROR := TRUE;
			AccessCase := 0;
		END_IF
		IF MachineWasRunning2 AND
			MachineMode2^.Auto AND
			NOT MachineMode2^.StopRequest AND
			NOT MachineMode2^.RapidStopRequest AND NOT LGVAccessActive THEN
				TFParametersArrayClear(ADR(ParametersArray));
				TFCommandSend(CmdDO,ParametersArray,MachineCmd2^);		
		ELSIF TFIsModuleError(MachineError2^) THEN
			AccessERRORCode := ErrMACHINEPALLETIZER_ERRORE_MACCHINA_IN_RICHIN;
			AccessERROR := TRUE;
			AccessCase := 0;
		END_IF
			
	61:	AccessReqIN := FALSE;
		AccessReqOUT := FALSE;
		AccessOK := FALSE;
		AccessCase := 0;
		MEMDiMarciaInPartenza := FALSE;
		
	ELSE
		AccessERROR := TRUE;
		AccessERRORCode := ErrMACHINEPALLETIZER_ERRORE_MACCHINA_IN_RICHIN;
		MEMDiMarciaInPartenza := FALSE;
		AccessCase := 0;
		
END_CASE

(* Clocks *)
IF TFTimerDone(ADR(Timer100)) THEN
	TFTimerSet(ADR(Timer100),100,TRUE);
	Clock100 := NOT Clock100;
END_IF
IF TFTimerDone(ADR(Timer500)) THEN
	TFTimerSet(ADR(Timer500),500,TRUE);
	Clock500 := NOT Clock500;
END_IF
IF TFTimerDone(ADR(Timer1000)) THEN
	TFTimerSet(ADR(Timer1000),1000,TRUE);
	Clock1000 := NOT Clock1000;
END_IF

(* Access Lamp *)
AccessLamp := 	(AccessOK OR
				(AccessReqOUT AND Clock500) OR
				(AccessReqIN AND Clock1000))AND
				NOT AccessERROR OR (AccessERROR AND Clock100);

END_FUNCTION_BLOCK

// ---- POUs/TFGateAccess/TFGateAccessNoStop.TcPOU
FUNCTION_BLOCK TFGateAccessNoStop
VAR_INPUT
	MachineCmd : POINTER TO CommandBuffer;
	MachineCmdExe : POINTER TO CommandExe;
	MachineState : POINTER TO State;
	MachineError : POINTER TO Error;
	MachineMode : POINTER TO Mode;
	Modules : POINTER TO TFPalletizerModules;
	Mission : POINTER TO TFMachinePalletizer_Mission;
	TimeBase : REAL;
	AccessRequest : BOOL;
	AccessDone : BOOL;
	LGVAccessActive	: BOOL;
	TilterPhaseStopDone : BOOL;
	PowerOK : BOOL;//Indica la presenza della marcia
	MacchinaInLavoroZonaOpposta : bool;//segnale da safety che indica che la macchina è in lavoro nella zona opposta a dove è stato effettuato l'ingresso... l'operatore può entrare senza far cadere la marcia
END_VAR
VAR_OUTPUT
	AccessLamp : BOOL; (* Access Lamp: 	OFF = No Access Consent,
										ON = Access Consent,
										FLASH (1sec) = Access Requested (Machine Stopping)
										FLASH (0.5sec) = Waiting Restart
										FLASH (0.1sec) = Access Error *)
										
	AccesActive : BOOL; (* Gate Acces Sequence in Execution *)
	AccessOK : BOOL;	(* Accesso consentito *)
	TilterPhaseStop : BOOL;		
	AccessERRORCode : UINT;		
	ErrAck : BOOL;
	ErrAckDriver : BOOL;			
END_VAR
VAR
	ParametersArray : ParametersArray;
	
	AccessERROR : BOOL;
	AccessReqIN : BOOL;
	AccessReqOUT : BOOL;
	AccessCase : INT;
	MachineWasRunning : BOOL;
	MachineWasRunning2 : bool;
	Timer100 : REAL;
	Timer500 : REAL;
	Timer1000 : REAL;
	Clock100 : BOOL;
	Clock500 : BOOL;
	Clock1000 : BOOL;
	TimerPowerOFF : real;
	MEMDiMarciaInPartenza : BOOL;
	TimerRitardoPower : REAL;
END_VAR

TFTimerCall(ADR(Timer100),TimeBase);
TFTimerCall(ADR(Timer500),TimeBase);
TFTimerCall(ADR(Timer1000),TimeBase);
TFTimerCall(ADR(TimerPowerOFF),TimeBase);
TFTimerCall(ADR(TimerRitardoPower),TimeBase);

CASE AccessCase OF
	
	(* Wait Request ON *)
	0:	AccesActive := FALSE;
		AccessOK := FALSE;
		AccessReqIN := FALSE;
		AccessReqOUT := FALSE;
		
		IF AccessRequest AND NOT AccessDone AND NOT TFIsModuleError(MachineError^) THEN
			//AccesActive := TRUE;
			AccessERROR := FALSE;
			AccessReqIN := TRUE;
			(* Machine Was Running if CmdDO and No Stop Request *) 
			MachineWasRunning := MachineCmdExe^.Code = CmdDO AND MachineCmdExe^.PhaseStopRequest = 0 AND MachineCmdExe^.RapidStopRequest = 0;
			IF MacchinaInLavoroZonaOpposta AND ((MachineWasRunning AND WorkAreaManager.State = WAMANAGER_NOP AND 
				TFPalletizerInPosizioneRiposo(ModuleAX_X:=ADR(Modules^.AX_X),ModuleAX_Y:=ADR(Modules^.AX_Y),ModuleAX_Z:=ADR(Modules^.AX_Z),ModuleAX_J:=ADR(Modules^.AX_J),Mission:=Mission)) OR
				NOT MachineWasRunning) THEN
					AccessCase := 25;
					AccesActive := TRUE;
			ELSIF TFIsModuleError(MachineError^) THEN
				AccessERRORCode := ErrMACHINEPALLETIZER_ERRORE_MACCHINA_IN_RICHIN;
				AccessERROR := TRUE;
				AccessCase := 0;
			END_IF
		ELSIF AccessERROR THEN
			AccessERRORCode := 0;
			AccessERROR 	:= FALSE;
			TilterPhaseStop := false;
		END_IF
		
	(* Access Ok.... Wait Request Done ON *)
	25:
		AccessReqIN 	:= FALSE;
		AccessReqOUT 	:= FALSE;
		AccessOK 		:= TRUE;
		IF NOT AccessRequest AND AccessDone THEN
			AccessCase := 27;
			TFTimerSet(ADR(TimerRitardoPower),100,TRUE);
			ErrAck := TRUE;
			//AccessOK 		:= FALSE;
			AccessReqOUT 	:= TRUE;
		END_IF
		IF TFIsModuleError(MachineError^) THEN
			AccessERRORCode := ErrMACHINEPALLETIZER_ERRORE_MACCHINA_IN_RICHIN;
			AccessERROR := TRUE;
			AccessCase := 0;
		END_IF
	
	(* *)	
	27:	IF NOT AccessDone THEN
			AccessCase := 28;
		END_IF
		
	(* *)	
	28:	IF AccessDone THEN
			AccessOK 		:= FALSE;
			AccessCase := 29;
		END_IF
	
	(* *)
	29:	IF NOT AccessDone THEN
			AccessCase := 60;
		END_IF

	(* Machine Restart *)
	60:	
		IF TFIsModuleError(MachineError^) THEN
			AccessERRORCode := ErrMACHINEPALLETIZER_ERRORE_MACCHINA_IN_RICHIN;
			AccessERROR := TRUE;
			AccessCase := 0;
		END_IF
		AccessCase := AccessCase + 1;
		
	(* *)
	61:	AccessReqIN := FALSE;
		AccessReqOUT := FALSE;
		AccessOK := FALSE;
		AccessCase := 0;
		MEMDiMarciaInPartenza := FALSE;
		
	ELSE
		AccessERROR := TRUE;
		AccessERRORCode := ErrMACHINEPALLETIZER_ERRORE_MACCHINA_IN_RICHIN;
		MEMDiMarciaInPartenza := FALSE;
		AccessCase := 0;
		
END_CASE

(* Clocks *)
IF TFTimerDone(ADR(Timer100)) THEN
	TFTimerSet(ADR(Timer100),100,TRUE);
	Clock100 := NOT Clock100;
END_IF
IF TFTimerDone(ADR(Timer500)) THEN
	TFTimerSet(ADR(Timer500),500,TRUE);
	Clock500 := NOT Clock500;
END_IF
IF TFTimerDone(ADR(Timer1000)) THEN
	TFTimerSet(ADR(Timer1000),1000,TRUE);
	Clock1000 := NOT Clock1000;
END_IF

(* Access Lamp *)
AccessLamp := 	((AccessOK AND NOT AccessReqOUT) OR
				(AccessReqOUT AND Clock1000) OR
				(AccessReqIN AND Clock1000))AND
				NOT AccessERROR OR (AccessERROR AND Clock100);

END_FUNCTION_BLOCK

// ---- POUs/TFLGV/TFLGV.TcPOU
FUNCTION_BLOCK TFLGV
VAR_INPUT
	WorkArea : POINTER TO ARRAY [1..MAXAREA] OF TFMachinePalletizer_WorkArea;
	WorkAreaState : POINTER TO ARRAY [1..MAXAREA] OF TFMachinePalletizer_WorkAreaState;
	PX_WorkArea : ARRAY [1..MAXAREA] OF BOOL;
	LGV_REQIN : BOOL;
	LGV_FOOTPRINT : BOOL;
	LGV_ReqIN_HW : BOOL;
	LGV_Footprint_HW : BOOL;
	LGV_ReqIN_SW : BOOL;
	LGV_Footprint_SW : BOOL;
	LGV_HW_SW_SWITCH : BOOL;
	MachineCmd : POINTER TO CommandBuffer;
	MachineCmdExe : POINTER TO CommandExe;
	MachineState : POINTER TO State;
	MachineError : POINTER TO Error;
	RobotError : POINTER TO Error;
	MachineMode : POINTER TO Mode;
	Power : BOOL;
	TimeBase : REAL;
	GateAccessActive : BOOL;
	ModuleAX_X : POINTER TO TFModulePalletizer_Ax;
	ModuleAX_Y : POINTER TO TFModulePalletizer_Ax;
	ModuleAX_Z : POINTER TO TFModulePalletizer_Ax;
	ModuleAX_J : POINTER TO TFModulePalletizer_Ax;
	ModuleAX_K : POINTER TO TFModulePalletizer_Ax;
	ModuloAsp  : POINTER TO	TFModulePalletizer_Aspirazione;
	Mission : POINTER TO TFMachinePalletizer_Mission;
	SecurityGateStatus : BOOL;
	ControlGateSecurity : POINTER TO BOOL;
	TilterPhaseStopDone : BOOL;	
END_VAR
VAR_OUTPUT
	LGV_Req : BOOL;
	LGV_LetIn : BOOL;
	LGVAccessLamp : BOOL; (* Access Lamp: 	OFF = No Access Consent,
										ON = Access Consent,
										FLASH (1sec) = Access Requested (Machine Stopping)
										FLASH (0.5sec) = Waiting Restart
										FLASH (0.1sec) = Access Error *)
										
	LGVAccesActive : BOOL; (* Gate Acces Sequence in Execution *)
	ClearWorkAreaLGVDone : BOOL;	
	TilterPhaseStop : BOOL;	
	LGVErrorCode : UINT;
	LGVResetHSKSUPNAV : BOOL;	
	LGV_ResetSW_RicIng : BOOL;
	LGVAccessOK : BOOL; (* Segnalazione accesso consentito *)
	ErrAck : BOOL; //Error Acknowledge Safaty
	ErrAckDriver : BOOL; //Error Acknowledge Drive
END_VAR
VAR
	LGVCase : INT;
	j : UINT;
	k : UINT; 
	
	ParametersArray : ParametersArray;
	//LGVAccessOK : BOOL;
	LGVAccessERROR : BOOL;	
	LGVAccessReqIN : BOOL;
	MachineWasRunning : BOOL;
	Timer100 : REAL;
	Timer200 : REAL;
	Timer1000 : REAL;
	Clock100 : BOOL;
	Clock200 : BOOL;
	Clock1000 : BOOL;
	TimerMachineWaitRunning : REAL;
	TimerPowerOFF : REAL;
	TimeoutControlloBarriereSicurezza : REAL;
	TimerOkBarriereSicurezze : REAL;
	TimeoutAnomaliaConsensi : REAL;
	TimerRitardoPower:REAL;
END_VAR

TFTimerCall(ADR(Timer100),TimeBase);
TFTimerCall(ADR(Timer200),TimeBase);
TFTimerCall(ADR(Timer1000),TimeBase);
TFTimerCall(ADR(TimerMachineWaitRunning),TimeBase);
TFTimerCall(ADR(TimerPowerOFF),TimeBase);
TFTimerCall(ADR(TimeoutControlloBarriereSicurezza),TimeBase);
TFTimerCall(ADR(TimerOkBarriereSicurezze),TimeBase);
TFTimerCall(ADR(TimeoutAnomaliaConsensi),TimeBase);
TFTimerCall(ADR(TimerRitardoPower),TimeBase);

IF LGV_HW_SW_SWITCH THEN
	LGV_REQIN := LGV_ReqIN_HW;
	LGV_FOOTPRINT := LGV_Footprint_HW;
ELSE	
	LGV_REQIN := LGV_ReqIN_SW;
	LGV_FOOTPRINT := LGV_Footprint_SW;
END_IF

LGV_Req := FALSE;
FOR j:=1 TO MAXAREA DO
	IF WorkAreaState^[j].State = WORKAREA_STATE_OCCUPIED_LGVREQ AND WorkArea^[j].Enable = 1 AND  WorkAreaState^[j].LGV_Req = 1 THEN
		LGV_Req := TRUE;
	END_IF
END_FOR

CASE LGVCase OF

	(* Case 0 *)
	0:	LGVErrorCode := 0;
		LGVResetHSKSUPNAV := false;
		LGVAccesActive := FALSE;
		LGVAccessOK := FALSE;
		LGVAccessReqIN := FALSE;
		TilterPhaseStop := FALSE;
		//LGV_Req := FALSE;
		(*FOR j:=1 TO MAXAREA DO
			IF WorkAreaState^[j].State = WORKAREA_STATE_OCCUPIED_LGVREQ AND WorkArea^[j].Enable = 1 AND  WorkArea^[j].LGV_Req = 1 THEN
				LGV_Req := TRUE;
			END_IF
		END_FOR*)
		
		// Command Case = 15 is WorkFlowsRunning after Homing WorkFlow NOTES: State=DO_RUN+1 it will be better!!!!
		MachineWasRunning := MachineCmdExe^.Code = CmdDO AND MachineCmdExe^.CmdCase = 15 AND MachineCmdExe^.PhaseStopRequest = 0 AND MachineCmdExe^.RapidStopRequest = 0;
		TFTimerSet(ADR(TimerMachineWaitRunning),1000,NOT MachineWasRunning);
		
		IF LGV_REQIN AND LGV_Req AND NOT GateAccessActive AND MachineWasRunning AND TFTimerDone(ADR(TimerMachineWaitRunning)) THEN
			LGVAccesActive := TRUE;
			LGVAccessERROR := FALSE;
			LGVAccessReqIN := TRUE;
			(* Machine Was Running if CmdDO and No Stop Request *)
			LGVCase := LGVCase + 1;
		END_IF	
			
	(* Case 1 - Phase Stop *)
	1:	TFParametersArrayClear(ADR(ParametersArray));
		TFCommandSend(CmdSTOPPHASE,ParametersArray,MachineCmd^);
		//TilterPhaseStop := TRUE;
		LGVCase := LGVCase + 1;
		
	(* Case 2 - Cmd DO END *)	
	2:	IF ((TFStateCodeGet(MachineState^) = StateDO_END AND NOT
			TFIsModuleError(MachineError^)) OR
			MachineCmdExe^.Code = CmdNOP)  THEN
			TilterPhaseStop := TRUE;
			TFTimerSet(ADR(TimerPowerOFF),1000,TRUE);
			LGVCase := LGVCase + 1;
		ELSIF TFIsModuleError(MachineError^) OR 
			ModuleAX_X^.Error.Code <> 0 OR
			ModuleAX_Y^.Error.Code <> 0 OR
			ModuleAX_Z^.Error.Code <> 0 OR
			ModuleAX_K^.Error.Code <> 0 OR
			ModuleAX_J^.Error.Code <> 0 OR
			ModuloAsp^.Error.Code <> 0 THEN
			LGVCase := 0; 
		END_IF

	(* Case 3 - Power Off *)
	3:	IF TFTimerDone(ADR(TimerPowerOFF)) AND TilterPhaseStopDone THEN
			TFParametersArrayClear(ADR(ParametersArray));
			ParametersArray.Parameters[0] := '0';
			TFCommandSend(CmdPOWER,ParametersArray,MachineCmd^);
			LGVCase := LGVCase + 1;
		END_IF	

	(* Case 4 - Power Off OK *)	
	4:	(*IF TFStateCodeGet(MachineState^) = StatePOWER_END OR
			TFIsModuleError(MachineError^) THEN
			LGVCase := LGVCase + 1;
		END_IF*)
		IF (TFStateCodeGet(MachineState^) = StatePOWER_END)AND// OR NOT Power) AND
			NOT TFIsModuleError(MachineError^) AND 
			NOT ModuleAX_X^.Error.Code <> 0 AND 
			NOT ModuleAX_Y^.Error.Code <> 0 AND
			NOT ModuleAX_Z^.Error.Code <> 0 AND
			NOT ModuleAX_K^.Error.Code <> 0 AND
			NOT ModuleAX_J^.Error.Code <> 0 AND
			NOT ModuloAsp^.Error.Code <> 0  AND 
			NOT GateAccessActive  AND TFPalletizerInPosizioneRiposo(ModuleAX_X,ModuleAX_Y,ModuleAX_Z,ModuleAX_J,Mission) THEN
			LGVCase := LGVCase + 1;
		ELSIF NOT LGV_REQIN THEN
			LGVCase := 6;
		ELSIF TFIsModuleError(MachineError^) OR 
			 (NOT TFPalletizerInPosizioneRiposo(ModuleAX_X,ModuleAX_Y,ModuleAX_Z,ModuleAX_J,Mission) AND (TFStateCodeGet(MachineState^) = StatePOWER_END OR NOT Power)) THEN
			LGVCase := 0;
		END_IF
		TFTimerSet(ADR(TimeoutAnomaliaConsensi),120000,TRUE);
		
	(* Case 5  LGV IN *)
	5:	
		IF LGV_REQIN AND LGV_Req AND NOT TFIsModuleError(MachineError^)THEN
			LGV_LetIn := TRUE;
			LGVAccessReqIN := FALSE;
			LGVAccessOK := TRUE;
			TFTimerSet(ADR(TimeoutAnomaliaConsensi),300000,TRUE);
		ELSIF TFIsModuleError(MachineError^) THEN // se la macchina è in errore, forzo l'uscita da questo stato
			LGV_ReqIN_SW := FALSE;
			LGV_Footprint_SW := FALSE;
			LGV_REQIN := LGV_ReqIN_SW;
			LGV_FOOTPRINT := LGV_Footprint_SW;
			LGVResetHSKSUPNAV := TRUE;
			LGVErrorCode := ErrMACHINEPALLETIZER_AZZERAMENTO_FORZATO_RICHIN_SUPNAVETTE;
			LGVCase := 0;
		ELSE
			LGV_LetIn := FALSE;
			LGVAccessOK := FALSE;
			LGVAccessReqIN := FALSE;
		END_IF
		
		IF NOT LGV_REQIN AND NOT LGV_FOOTPRINT THEN
			LGV_LetIn := FALSE;
			LGVCase := LGVCase + 1;
		ELSIF TFTimerDone(ADR(TimeoutAnomaliaConsensi)) AND ((LGV_REQIN AND NOT LGV_FOOTPRINT) OR (NOT LGV_REQIN AND LGV_FOOTPRINT)) THEN
			LGV_ReqIN_SW := FALSE;
			LGV_Footprint_SW := FALSE;
			LGV_REQIN := LGV_ReqIN_SW;
			LGV_FOOTPRINT := LGV_Footprint_SW;
			LGVResetHSKSUPNAV := TRUE;
			LGVErrorCode := ErrMACHINEPALLETIZER_ANOMALIA_CONSENSI_SUPNAVETTE;
			LGVCase := 0;
		ELSIF TFIsModuleError(MachineError^) THEN // se la macchina è in errore, forzo l'uscita da questo stato
			LGV_ReqIN_SW := FALSE;
			LGV_Footprint_SW := FALSE;
			LGV_REQIN := LGV_ReqIN_SW;
			LGV_FOOTPRINT := LGV_Footprint_SW;
			LGVResetHSKSUPNAV := TRUE;
			LGVErrorCode := ErrMACHINEPALLETIZER_AZZERAMENTO_FORZATO_RICHIN_SUPNAVETTE;
			LGVCase := 0;
		END_IF	
		TFTimerSet(ADR(TimeoutControlloBarriereSicurezza),20000,TRUE);

	(* Case 6 - Clear / Setup WorkArea *)
	6:	
		FOR k:= 1 TO 6 DO
			IF NOT PX_WorkArea[k] (*OR 
				(WorkAreaState^[k].State = WORKAREA_STATE_OCCUPIED_LGVREQ AND WorkArea^[k].Enable = 1 AND  WorkArea^[k].LGV_Req = 1)*) THEN
				// Pulisco piazzola in seguito ad estrazione
				TFClearWorkArea(WorkArea,WorkAreaState,k);
				I_PHPresenzaPalletVirtuale[k]:=FALSE;
			ELSE
				// preparo la piazzola solo se di tipo catasta pallet o layer	
				//IF WorkArea^[k].Typology = TYPOLOGY_STACK OR WorkArea^[k].Typology = TYPOLOGY_LAYER THEN
				//	TFClearWorkAreaStack(WorkArea,WorkAreaState,k);
				;//END_IF
			END_IF
		END_FOR
		LGVCase := LGVCase + 1;	
		
		
		IF TFIsModuleError(MachineError^) THEN // se la macchina è in errore, forzo l'uscita da questo stato
			LGV_ReqIN_SW := FALSE;
			LGV_Footprint_SW := FALSE;
			LGV_REQIN := LGV_ReqIN_SW;
			LGV_FOOTPRINT := LGV_Footprint_SW;
			LGVResetHSKSUPNAV := TRUE;
			LGVErrorCode := ErrMACHINEPALLETIZER_AZZERAMENTO_FORZATO_RICHIN_SUPNAVETTE;
			LGVCase := 0;
		END_IF
	
	7:
		FOR k:= 6 TO MAXAREAPRESENT DO
			IF NOT PX_WorkArea[k] (*OR 
				(WorkAreaState^[k].State = WORKAREA_STATE_OCCUPIED_LGVREQ AND WorkArea^[k].Enable = 1 AND  WorkArea^[k].LGV_Req = 1)*) THEN
				// Pulisco piazzola in seguito ad estrazione
				TFClearWorkArea(WorkArea,WorkAreaState,k);
				I_PHPresenzaPalletVirtuale[k]:=FALSE;
			ELSE
				// preparo la piazzola solo se di tipo catasta pallet o layer	
				//IF WorkArea^[k].Typology = TYPOLOGY_STACK OR WorkArea^[k].Typology = TYPOLOGY_LAYER THEN
				//	TFClearWorkAreaStack(WorkArea,WorkAreaState,k);
				;//END_IF
			END_IF
		END_FOR
		ClearWorkAreaLGVDone := TRUE;
		LGVAccessOK := FALSE;
		LGVCase := 10;	
		TFTimerSet(ADR(TimerOkBarriereSicurezze),1000, TRUE);	
		IF TFIsModuleError(MachineError^) THEN // se la macchina è in errore, forzo l'uscita da questo stato
			LGV_ReqIN_SW := FALSE;
			LGV_Footprint_SW := FALSE;
			LGV_REQIN := LGV_ReqIN_SW;
			LGV_FOOTPRINT := LGV_Footprint_SW;
			LGVResetHSKSUPNAV := TRUE;
			LGVErrorCode := ErrMACHINEPALLETIZER_AZZERAMENTO_FORZATO_RICHIN_SUPNAVETTE;
			LGVCase := 0;
		END_IF
		
	(* Case 7 - Power ON *)
	10:	//TFTimerSet(ADR(TimerOkBarriereSicurezze),5000, NOT SecurityGateStatus);
		IF NOT GateAccessActive AND TFTimerDone(ADR(TimerOkBarriereSicurezze))  THEN
			TFTimerSet(ADR(TimerRitardoPower),100,TRUE);
			LGVCase := LGVCase + 1;	
		ELSIF TFTimerDone(ADR(TimeoutControlloBarriereSicurezza)) THEN
			LGVErrorCode := ErrMACHINEPALLETIZER_BARRIEREOCCUPATE_LGVREQ_OFF;
			LGVCase := 0;
		ELSIF TFIsModuleError(MachineError^) THEN // se la macchina è in errore, forzo l'uscita da questo stato
			LGV_ReqIN_SW := FALSE;
			LGV_Footprint_SW := FALSE;
			LGV_REQIN := LGV_ReqIN_SW;
			LGV_FOOTPRINT := LGV_Footprint_SW;
			LGVResetHSKSUPNAV := TRUE;
			LGVErrorCode := ErrMACHINEPALLETIZER_AZZERAMENTO_FORZATO_RICHIN_SUPNAVETTE;
			LGVCase := 0;
		END_IF
(**************************************************************************)
(**************** Error Acknowledge Safety + AZIONAMENTI ***************************)
	11:
		IF TFTimerDone(ADR(TimerRitardoPower)) THEN
			TFTimerSet(ADR(TimerRitardoPower),100,TRUE);
			ErrAck := TRUE;
			LGVCase := LGVCase + 1;	
		END_IF
		
	12:	
		IF TFTimerDone(ADR(TimerRitardoPower)) THEN
			TFTimerSet(ADR(TimerRitardoPower),100,TRUE);
			ErrAck := FALSE;
			LGVCase := LGVCase + 1;	
		END_IF

	13:
		IF TFTimerDone(ADR(TimerRitardoPower)) THEN
			TFTimerSet(ADR(TimerRitardoPower),100,TRUE);
			ErrAckDriver := TRUE;
			LGVCase := LGVCase+1;
		END_IF
		
	14:
		IF TFTimerDone(ADR(TimerRitardoPower)) THEN
			TFTimerSet(ADR(TimerRitardoPower),100,TRUE);
			ErrAckDriver := FALSE;
			LGVCase := LGVCase+1;
		END_IF

	15: IF TFTimerDone(ADR(TimerRitardoPower)) THEN
			LGVCase := 20;
		END_IF
(**************************************************************************)
(**************************************************************************)		
	(* Case 20 - Power ON *)
	20:	//TFTimerSet(ADR(TimerOkBarriereSicurezze),5000, NOT SecurityGateStatus);
		IF NOT GateAccessActive AND TFTimerDone(ADR(TimerOkBarriereSicurezze))  THEN
			TFParametersArrayClear(ADR(ParametersArray));
			ParametersArray.Parameters[0] := '1';
			TFCommandSend(CmdPOWER,ParametersArray,MachineCmd^);
			LGV_ResetSW_RicIng := TRUE;
			LGVCase := LGVCase + 1;	
		ELSIF TFTimerDone(ADR(TimeoutControlloBarriereSicurezza)) THEN
			LGVErrorCode := ErrMACHINEPALLETIZER_BARRIEREOCCUPATE_LGVREQ_OFF;
			LGVCase := 0;
		END_IF	
			
	(* Case 21 - Power On OK *)
	21:	IF TFStateCodeGet(MachineState^) = StatePOWER_END OR
			TFIsModuleError(MachineError^) THEN
			LGV_ResetSW_RicIng := FALSE;
			LGVCase := LGVCase + 1;	
		END_IF
		
	(* Case 22 - Cmd DO *)
	22:	
		IF MachineWasRunning AND
			MachineMode^.Auto AND
			NOT MachineMode^.StopRequest AND
			NOT MachineMode^.RapidStopRequest AND NOT GateAccessActive THEN
			(*AND (SecurityGateStatus OR NOT ControlGateSecurity^*) 
			TFParametersArrayClear(ADR(ParametersArray));
			TFCommandSend(CmdDO,ParametersArray,MachineCmd^);
			TilterPhaseStop := FALSE;
		END_IF
		LGVCase := 0;
	
	ELSE
		LGVAccessERROR := TRUE;
		LGVCase := 0;
	
END_CASE

(* Clocks *)
IF TFTimerDone(ADR(Timer100)) THEN
	TFTimerSet(ADR(Timer100),100,TRUE);
	Clock100 := NOT Clock100;
END_IF
IF TFTimerDone(ADR(Timer200)) THEN
	TFTimerSet(ADR(Timer200),200,TRUE);
	Clock200 := NOT Clock200;
END_IF
IF TFTimerDone(ADR(Timer1000)) THEN
	TFTimerSet(ADR(Timer1000),1000,TRUE);
	Clock1000 := NOT Clock1000;
END_IF

(* Access Lamp *)
LGVAccessLamp := ((LGVAccessOK AND Clock200) OR
				//(AccessReqOUT AND Clock500) OR
				(LGVAccessReqIN AND Clock1000))AND
				NOT LGVAccessERROR OR (LGVAccessERROR AND Clock100);

END_FUNCTION_BLOCK

// ---- POUs/TFPalletizerData/TFClearWorkArea.TcPOU
FUNCTION TFClearWorkArea : BOOL
VAR_INPUT
	WorkArea : POINTER TO  TFMachinePalletizer_WorkArea;
	WorkAreaState : POINTER TO TFMachinePalletizer_WorkAreaState;
END_VAR
VAR

END_VAR

WorkAreaState^ 				:= EmptyWorkAreaState;
WorkAreaState^.State		:= WORKAREA_STATE_FREE_ENABLED;	(* Stato Area di Lavoro/Piazzola
																			(0=Assente e Area Disabilitata,
																			1=Presente e Area Disabilitata,
																			2=Assente in Lavorazione,
																			3=Presente in Lavorazione,
																			4=Presente con Pallettizzazione Terminata,
																			5=Presente con Pallettizzazione Terminata e Area Disabilitata,
																			6=Presente in Nastratura,
																			7=Presente in Nastratura e Area Disabilitata,
																			8=Presente con Nastratura Terminata,
																			9=Presente con Nastratura Terminata e Area Disabilitata,
																			10=Presente con Lavorazione Terminata,
																			11=Presente con Lavorazione Terminata e Area Disabilitata,
																			12=Presente con LGV in Richiesta Ingresso,
																			13=Presente con LGV in Richiesta Ingresso e Area Disabilitata,
																			14=Presente con LGV in Ingombro,
																			15=Presente con LGV in Ingombro e Area Disabilitata,
																			16=Presente con LGV Fuori Ingombro e Pallet Estratto,
																			17=Presente con LGV Fuori Ingombro e Pallet Estratto e Area Disabilitata, NOT USED !!!!!!!!!!!
																			99=Errore
																			-1 dato non valido) *)
WorkAreaState^.F					:= 0;	(* Forming Pointer - Puntatore tabella formature (1..n=, -1 dato non valido *)
WorkAreaState^.P					:= 1;	(* Pack Pointer - Puntatore tabella ELEMENTO (0..n-1=, -1 dato non valido),Numero ELEMENTO successivo da depositare *)
WorkAreaState^.P_Cava.HMI_NumeroPezziPresentiPostazione_A_Cavaleto		:= 1 ;
WorkAreaState^.P_Cava.HMI_NumeroPezziPresentiPostazione_B_Cavaleto		:= 1 ;

              
WorkAreaState^.Code					:= 0;	(* Codice di Pallettizzazione (0..n=, -1 dato non valido) x lastre, se Magazzino Falde, codice della falda *)
              
WorkAreaState^.PackPointerModified	:= FALSE;		(* Se TRUE, indica che è stata effettuata una modfica sui dati della WA da parte dell' HMI (Settata da HMI e resettata da PLC) *)
WorkAreaState^.PackPointer			:= 0;			(* Rappresenta l'indice del pacco da depositare dopo modfica manuale,cioè con PackPointerModified=TRUE *)

WorkAreaState^.Slab := EmptySlabArray;

WorkAreaState^.LGVAttr				:= 0;

TFClearWorkAreaBCRead(WorkAreaState);//Resetto i vari stati dl BARCODE

WorkAreaState^.H					:= 0.0; (* (mm) Altezza Reale. Viene calcolata dal PLC dopo ogni prelievo (Vuoti o Falde) o deposito Pallet e durante la pallettizzazione *)
WorkAreaState^.HPL					:= 0.0; (* (mm) Altezza del pallett utilizzato + altezza layers utilizzati *)

TFClearApprendimento(ADR(WorkAreaState^.Apprendimento));//Azzeramento apprendimento

(*
(* Apprendimenti nelle varie direzioni *)
WorkAreaState^[k].DoLearn_Y0		:= APPRENDIMENTO_DA_ESEGUIRE;	(* Stato apprendimento Direzione Y LATO 0° 0=Disabilitato, 1=Abilitato da Eseguire, 2=Eseguito, -1 dato non valido *)
WorkAreaState^[k].Learn_Y0			:= 0.0;	(* (mm) Quota inizio Apprendimento Direzione Y LATO 0° *)
WorkAreaState^[k].Learned_Y0		:= 0.0; (* Quota rilevata durante apprendimento Direzione Y LATO 0° *)

WorkAreaState^[k].DoLearn_Y180		:= APPRENDIMENTO_DA_ESEGUIRE;	(* Stato apprendimento Direzione Y LATO 180° 0=Disabilitato, 1=Abilitato da Eseguire, 2=Eseguito, -1 dato non valido *)
WorkAreaState^[k].Learn_Y180		:= 0.0;	(* (mm) Quota inizio Apprendimento Direzione Y LATO 180° *)
WorkAreaState^[k].Learned_Y180		:= 0.0; (* Quota rilevata durante apprendimento Direzione Y LATO 180° *)

WorkAreaState^[k].DoLearn_Z			:= APPRENDIMENTO_DA_ESEGUIRE;	(* Stato apprendimento Direzione Z 0=Disabilitato, 1=Abilitato da Eseguire, 2=Eseguito, -1 dato non valido *)
WorkAreaState^[k].Learn_Z			:= 0.0;	(* (mm) Quota inizio Apprendimento Direzione Z *)
WorkAreaState^[k].Learned_Z			:= 0.0; (* Quota rilevata durante apprendimento Direzione Z *)
*)
WorkAreaState^.RefuseLGV       	:= FALSE;	(* Abilitazione chiamata LGV a termine pallettizzazione - TRUE= Non chiama LGV quando pallet pieno, FALSE= viene eseguita richiesta LGV *)
              
WorkAreaState^.LGV_Req			:= 0;	(* Richiesta LGV (0=Nop, 1=Richiesta LGV, 2= Consenso Ingresso, -1= non valido) *)
WorkAreaState^.LGV_GetIn_GetOut	:= 0;	(* Tipo Richiesta LGV  (0=Nop, 1=Richiesta Prelievo, 2= Richiesta Deposito, -1= non valido) *)	
WorkAreaState^.LGV_ReqAbort		:= FALSE; (* Aborto chimata LGV *)

WorkAreaState^.SlabData := EmptyDataSlabArray;

TFClearWorkArea := TRUE;

END_FUNCTION

// ---- POUs/TFLGV/TFLGV_NEW.TcPOU
FUNCTION_BLOCK TFLGV_NEW
VAR_INPUT
	WorkArea : POINTER TO ARRAY [1..MAXAREA] OF TFMachinePalletizer_WorkArea;
	WorkAreaState : POINTER TO ARRAY [1..MAXAREA] OF TFMachinePalletizer_WorkAreaState;
	PH_WorkArea : ARRAY [1..MAXAREA] OF BOOL;

	MachineCmd : POINTER TO CommandBuffer;
	MachineCmdExe : POINTER TO CommandExe;
	MachineState : POINTER TO State;
	MachineError : POINTER TO Error;
	RobotError : POINTER TO Error;
	MachineMode : POINTER TO Mode;
	Power : BOOL;
	TimeBase : REAL;
	GateAccessActive : BOOL;
	ModuleAX_X : POINTER TO TFModulePalletizer_Ax;
	ModuleAX_Y : POINTER TO TFModulePalletizer_Ax;
	ModuleAX_Z : POINTER TO TFModulePalletizer_Ax;
	ModuleAX_J : POINTER TO TFModulePalletizer_Ax;
	ModuleAX_K : POINTER TO TFModulePalletizer_Ax;
	ModuloAsp  : POINTER TO	TFModulePalletizer_Aspirazione;
	Mission : POINTER TO TFMachinePalletizer_Mission;
	BarriereSicurezzaEsterneOK : BOOL; // Stato delle barriere di sicurezza, TRUE=Barriere OK 
	ControlGateSecurity : POINTER TO BOOL;
	TilterPhaseStopDone : BOOL;	
	
	LGV_Stato_Operazione  : POINTER TO ARRAY [1..MAXAREA] OF e_Stato_Operazione_LGV; // Indica lo stato dell'operazione svolta dalla navetta: 0=Dato ricevuto e azzerato da PLC,1= Deposito Concluso,2= Prelievo Concluso,
	LGV_RichiestaIngresso : ARRAY [1..MAXAREA] OF BOOL; 	// Chiamata ingresso DA LGV,TRUE= La postazione è nello stato di chiamata navetta
	LGV_InIngombro		  : ARRAY [1..MAXAREA] OF BOOL; 	// Segnale di LGV in ingombro da supervisione navette 
	
END_VAR
VAR_OUTPUT
	
	LGV_ChiamataDaPostazione	: ARRAY [1..MAXAREA] OF BOOL; 	// Chiamata ingresso a LGV,TRUE=La una postazione è nello stato di chiamata navetta
	LGV_OkIngressoInPostazione 	: ARRAY [1..MAXAREA] OF BOOL; 	// TRUE = OK Ingresso Nella Postazione 
	
	MEM_LGV_InIngombro		  : ARRAY [1..MAXAREA] OF BOOL; 	// Memoria LGV in INGOMBRO

	
	LGVAccessLamp : BOOL; (* Access Lamp: 	OFF = No Access Consent,
										ON = Access Consent,
										FLASH (1sec) = Access Requested (Machine Stopping)
										FLASH (0.5sec) = Waiting Restart
										FLASH (0.1sec) = Access Error *)
										
	LGVAccesActive : BOOL; (* Gate Acces Sequence in Execution *)
	ClearWorkAreaLGVDone : BOOL;	
	TilterPhaseStop : BOOL;	
	LGVErrorCode : UINT;
	LGVResetHSKSUPNAV : BOOL;	
	LGV_ResetSW_RicIng : BOOL;
	LGVAccessOK : BOOL; (* Segnalazione accesso consentito *)
END_VAR
VAR
	LGVCase : INT;
	j : UINT;
	k : UINT; 
	i : UINT;
	
	ParametersArray : ParametersArray;
	
	LGVAccessERROR : BOOL;	
	LGVAccessReqIN : ARRAY [1..MAXAREA] OF BOOL;
	MachineWasRunning : BOOL;
	Timer100 : REAL;
	Timer200 : REAL;
	Timer1000 : REAL;
	Clock100 : BOOL;
	Clock200 : BOOL;
	Clock1000 : BOOL;
	TimerMachineWaitRunning : REAL;
	TimerPowerOFF : REAL;
	TimeoutControlloBarriereSicurezza : REAL;
	TimerOkBarriereSicurezze : REAL;
	TimeoutAnomaliaConsensi : REAL;
	LampadaIngressoInCorso : BOOL;//Se almeno una postazione è in chiamata e la navetta ha fatto la richiesta di ingresso
	iPost:UINT;
	iRichIngr:INT;
END_VAR

TFTimerCall(ADR(Timer100),TimeBase);
TFTimerCall(ADR(Timer200),TimeBase);
TFTimerCall(ADR(Timer1000),TimeBase);
TFTimerCall(ADR(TimerMachineWaitRunning),TimeBase);
TFTimerCall(ADR(TimerPowerOFF),TimeBase);
TFTimerCall(ADR(TimeoutControlloBarriereSicurezza),TimeBase);
TFTimerCall(ADR(TimerOkBarriereSicurezze),TimeBase);
TFTimerCall(ADR(TimeoutAnomaliaConsensi),TimeBase);

(* Setto lo stato della chiamata *)
FOR j:=1 TO MAXAREAPRESENT DO
	IF WorkAreaState^[j].State = WORKAREA_STATE_OCCUPIED_LGVREQ AND WorkArea^[j].Enable = 1 AND  WorkAreaState^[j].LGV_Req = 1 THEN
		LGV_ChiamataDaPostazione[j] := TRUE;
	ELSE
		LGV_ChiamataDaPostazione[j] := FALSE;
	END_IF
END_FOR

CASE LGVCase OF

	(* Case 0 *)
	0:	LGVErrorCode := 0;
		LGVResetHSKSUPNAV := false;
		LGVAccesActive := FALSE;
		LGVAccessOK := FALSE;
		TilterPhaseStop := FALSE;
		LampadaIngressoInCorso := FALSE;		
		(* Se la macchina è in automatico da almeno un minuto verifico se ho una richiesta di ingresso e in questo caso attivo la procedura di richiesta ingresso *)
		MachineWasRunning := MachineCmdExe^.Code = CmdDO AND MachineCmdExe^.CmdCase = 15 AND MachineCmdExe^.PhaseStopRequest = 0 AND MachineCmdExe^.RapidStopRequest = 0;
		TFTimerSet(ADR(TimerMachineWaitRunning),1000,NOT MachineWasRunning);
		FOR i:=1 TO MAXAREAPRESENT DO
			IF LGV_RichiestaIngresso[i] AND //Richiesta ingresso DA NAVETTA
				LGV_ChiamataDaPostazione[i] AND //Piazzola in Chiamata
				NOT GateAccessActive AND //Richiesta di ingresso manuale NON ATTIVA
				MachineWasRunning AND TFTimerDone(ADR(TimerMachineWaitRunning)) THEN //Macchina in automatico e senza errori per almeno un minuto
					LGVAccesActive := TRUE; 	//Setto lo stato di richiesta ingresso in corso
					LGVAccessERROR := FALSE;	//Resetto la memoria di errore durante una richiesta di ingresso
					LGVAccessReqIN[i] := TRUE;	//Setto una memoria che mi indica quale sia la postazione che ha fatto la richiesta
					LampadaIngressoInCorso := TRUE; //Lampada di segnalazione
					LGVCase := LGVCase + 1;		//Vado allo stato successivo
					EXIT;
			ELSE
				LGVAccessReqIN[i] := FALSE; 	//Resetto lo stato di richiesta ingresso in corso
			END_IF	
		END_FOR
			
	(* Case 1 - Lancio lo stop in fase del pallettizzatore *)
	1:	TFParametersArrayClear(ADR(ParametersArray));
		TFCommandSend(CmdSTOPPHASE,ParametersArray,MachineCmd^);
		LGVCase := LGVCase + 1;
		
	(* Case 2 - Attendo che lo stop in fase sia avvenuto *)	
	2:	IF ((TFStateCodeGet(MachineState^) = StateDO_END AND 
			NOT TFIsModuleError(MachineError^)) OR
			MachineCmdExe^.Code = CmdNOP)  THEN
				TilterPhaseStop := TRUE;
				TFTimerSet(ADR(TimerPowerOFF),1000,TRUE);
				LGVCase := LGVCase + 1;
		ELSIF TFIsModuleError(MachineError^) OR 
			ModuleAX_X^.Error.Code <> 0 OR
			ModuleAX_Y^.Error.Code <> 0 OR
			ModuleAX_Z^.Error.Code <> 0 OR
			ModuleAX_K^.Error.Code <> 0 OR
			ModuleAX_J^.Error.Code <> 0 OR
			ModuloAsp^.Error.Code <> 0 THEN
			LGVCase := 0; 
		END_IF

	(* Case 3 - Richiesta di Power Off *)
	3:	IF TFTimerDone(ADR(TimerPowerOFF)) THEN//AND TilterPhaseStopDone THEN
			TilterPhaseStop := FALSE;
			TFParametersArrayClear(ADR(ParametersArray));
			ParametersArray.Parameters[0] := '0';
			TFCommandSend(CmdPOWER,ParametersArray,MachineCmd^);
			LGVCase := LGVCase + 1;
		END_IF	

	(* Case 4 - Power Off OK *)	
	4:	
		TFTimerSet(ADR(TimeoutAnomaliaConsensi),120000,TRUE);
		IF (TFStateCodeGet(MachineState^) = StatePOWER_END OR NOT Power) AND
			NOT TFIsModuleError(MachineError^) AND 
			NOT ModuleAX_X^.Error.Code <> 0 AND 
			NOT ModuleAX_Y^.Error.Code <> 0 AND
			NOT ModuleAX_Z^.Error.Code <> 0 AND
			NOT ModuleAX_K^.Error.Code <> 0 AND
			NOT ModuleAX_J^.Error.Code <> 0 AND
			NOT ModuloAsp^.Error.Code <> 0  AND 
			NOT GateAccessActive  AND 
			TFPalletizerInPosizioneRiposo(ModuleAX_X,ModuleAX_Y,ModuleAX_Z,ModuleAX_J,Mission) THEN
				LGVCase := LGVCase + 1;
		ELSIF TFIsModuleError(MachineError^) OR 
			 (NOT TFPalletizerInPosizioneRiposo(ModuleAX_X,ModuleAX_Y,ModuleAX_Z,ModuleAX_J,Mission) AND (TFStateCodeGet(MachineState^) = StatePOWER_END OR NOT Power)) THEN
			LGVCase := 0;
		END_IF
		
	(* Case 5 - Guardo se la postazione è in chiamata *)
	5:	
		TFTimerSet(ADR(TimeoutControlloBarriereSicurezza),20000,TRUE);
		TFTimerSet(ADR(TimeoutAnomaliaConsensi),120000,((LGV_RichiestaIngresso[iPost] AND NOT LGV_InIngombro[iPost]) OR (NOT LGV_RichiestaIngresso[iPost] AND LGV_InIngombro[iPost])));		//Setto il timer per la rilevazione di eventuali anomalie nello scambio consensi

		IF NOT TFIsModuleError(MachineError^) THEN //Se la macchina NON è in errore 
			FOR iPost:=1 TO MAXAREAPRESENT DO	//Ciclo tutte le postazioni
				IF LGV_ChiamataDaPostazione[iPost] AND LGV_RichiestaIngresso[iPost] AND NOT LGV_OkIngressoInPostazione[iPost] THEN //Se ho la postazione in chiamata e la richiesta di ingresso corrispondente PROCEDO con il ciclo
					LGVAccessOK := TRUE;										//Setto memoria per gestione lampada
					LGV_OkIngressoInPostazione[iPost] := TRUE;					//Setto a TRUE l'ok all'ingresso della postazione designata
				ELSIF LGV_ChiamataDaPostazione[iPost] AND NOT LGV_RichiestaIngresso[iPost] AND LGV_OkIngressoInPostazione[iPost] THEN //Se HO la postazione in chiamata e è CADUTA la richiesta di ingresso alla postazione genero ERRORE e esco
					LGVAccessOK := FALSE;
					LGV_OkIngressoInPostazione[iPost] := FALSE;
					LGVErrorCode := ErrMACHINEPALLETIZER_PERDITARICHIAMATAPOST;	
					LGVCase := 0;
				ELSIF NOT LGV_ChiamataDaPostazione[iPost] AND LGV_RichiestaIngresso[iPost] AND LGV_OkIngressoInPostazione[iPost] THEN //Se NON ho la postazione in chiamata e HO la richiesta di ingresso alla postazione genero ERRORE e esco
					LGVAccessOK := FALSE;
					LGV_OkIngressoInPostazione[iPost] := FALSE;
					LGVErrorCode := ErrMACHINEPALLETIZER_PERDITARICINGRESSOPOST;
					LGVCase := 0;
				ELSE
					;
				END_IF
	
				(* Setto la memoria che mi indica che la navetta ha segnalato l'ingombro *)
				IF LGV_OkIngressoInPostazione[iPost] AND LGV_RichiestaIngresso[iPost] AND LGV_InIngombro[iPost] THEN
					MEM_LGV_InIngombro[iPost]:=TRUE;
				END_IF
						
				(* Attendo che la navetta abbia finito il suo ciclo. Proseguo al riavvio della macchina SOLO quando mi cadono la richiesta di ingresso e l'ingombro *)
				IF MEM_LGV_InIngombro[iPost] THEN
					IF NOT LGV_RichiestaIngresso[iPost] AND NOT LGV_InIngombro[iPost] THEN //Se non ho più la richiesta di ingresso e ho NON HO PIU' l'ingombro della navetta, proseguo con il ciclo di restar macchina
						MEM_LGV_InIngombro[iPost]:=FALSE;
						LGVCase := LGVCase + 1;
					ELSIF TFTimerDone(ADR(TimeoutAnomaliaConsensi)) THEN//((LGV_RichiestaIngresso[iPost] AND NOT LGV_InIngombro[iPost]) OR (NOT LGV_RichiestaIngresso[iPost] AND LGV_InIngombro[iPost])) THEN
						LGVErrorCode := ErrMACHINEPALLETIZER_ANOMALIA_CONSENSI_SUPNAVETTE;
						LGVCase := 0;
					END_IF
				END_IF
		
			END_FOR
		ELSE							//Se la macchina è in ERRORE
			LGVErrorCode := ErrMACHINEPALLETIZER_AZZERAMENTO_FORZATO_RICHIN_SUPNAVETTE;
		END_IF
	
	(*
		IF LGV_RichiestaIngresso[i] AND LGV_ChiamataDaPostazione[i] AND NOT TFIsModuleError(MachineError^)THEN
			LGV_LetIn := TRUE;
			LGVAccessReqIN := FALSE;
			LGVAccessOK := TRUE;
			TFTimerSet(ADR(TimeoutAnomaliaConsensi),120000,TRUE);
		ELSIF TFIsModuleError(MachineError^) THEN // se la macchina è in errore, forzo l'uscita da questo stato
			LGV_ReqIN_SW := FALSE;
			LGV_Footprint_SW := FALSE;
			LGV_REQIN := LGV_ReqIN_SW;
			LGV_FOOTPRINT := LGV_Footprint_SW;
			LGVResetHSKSUPNAV := TRUE;
			LGVErrorCode := ErrMACHINEPALLETIZER_AZZERAMENTO_FORZATO_RICHIN_SUPNAVETTE;
			LGVCase := 0;
		ELSE
			LGV_LetIn := FALSE;
			LGVAccessOK := FALSE;
			LGVAccessReqIN := FALSE;
		END_IF
		
		IF NOT LGV_REQIN AND NOT LGV_FOOTPRINT THEN
			LGV_LetIn := FALSE;
			LGVCase := LGVCase + 1;
		ELSIF TFTimerDone(ADR(TimeoutAnomaliaConsensi)) AND ((LGV_REQIN AND NOT LGV_FOOTPRINT) OR (NOT LGV_REQIN AND LGV_FOOTPRINT)) THEN
			LGV_ReqIN_SW := FALSE;
			LGV_Footprint_SW := FALSE;
			LGV_REQIN := LGV_ReqIN_SW;
			LGV_FOOTPRINT := LGV_Footprint_SW;
			LGVResetHSKSUPNAV := TRUE;
			LGVErrorCode := ErrMACHINEPALLETIZER_ANOMALIA_CONSENSI_SUPNAVETTE;
			LGVCase := 0;
		END_IF	*)
		

	(* Case 6 - Clear / Setup WorkArea *)
	6:	
	
